LIN {X 0,Y 523.917,Z 214.223,A -85,B 0,C 180,E1 -4816.833,E2 -4816.833} C_VEL
LIN {X 0,Y 523.939,Z 214.219,A -85,B 0,C 180,E1 -4818.907,E2 -4818.907} C_VEL
LIN {X 0,Y 523.916,Z 214.219,A -85,B 0,C 180,E1 -4821.898,E2 -4821.898} C_VEL
LIN {X 0,Y 523.935,Z 214.221,A -85,B 0,C 180,E1 -4824.909,E2 -4824.909} C_VEL
LIN {X 0,Y 523.935,Z 214.217,A -85,B 0,C 180,E1 -4827.68,E2 -4827.68} C_VEL
LIN {X 0,Y 523.954,Z 214.217,A -85,B 0,C 180,E1 -4830.676,E2 -4830.676} C_VEL
LIN {X 0,Y 523.973,Z 214.213,A -85,B 0,C 180,E1 -4833.728,E2 -4833.728} C_VEL
LIN {X 0,Y 523.925,Z 214.217,A -85,B 0,C 180,E1 -4836.27,E2 -4836.27} C_VEL
LIN {X 0,Y 523.945,Z 214.22,A -85,B 0,C 180,E1 -4838.767,E2 -4838.767} C_VEL
LIN {X 0,Y 523.948,Z 214.219,A -85,B 0,C 180,E1 -4841.221,E2 -4841.221} C_VEL
LIN {X 0,Y 523.935,Z 214.217,A -85,B 0,C 180,E1 -4843.639,E2 -4843.639} C_VEL
LIN {X 0,Y 523.939,Z 214.213,A -85,B 0,C 180,E1 -4846.028,E2 -4846.028} C_VEL
LIN {X 0,Y 524.012,Z 214.209,A -85,B 0,C 180,E1 -4848.394,E2 -4848.394} C_VEL
LIN {X 0,Y 524.003,Z 214.209,A -85,B 0,C 180,E1 -4851.516,E2 -4851.516} C_VEL
LIN {X 0,Y 524.08,Z 214.203,A -85,B 0,C 180,E1 -4854.614,E2 -4854.614} C_VEL
LIN {X 0,Y 524.111,Z 214.195,A -85,B 0,C 180,E1 -4857.695,E2 -4857.695} C_VEL
LIN {X 0,Y 524.123,Z 214.199,A -85,B 0,C 180,E1 -4860.768,E2 -4860.768} C_VEL
LIN {X 0,Y 524.069,Z 214.203,A -85,B 0,C 180,E1 -4863.075,E2 -4863.075} C_VEL
LIN {X 0,Y 524.035,Z 214.205,A -85,B 0,C 180,E1 -4866.159,E2 -4866.159} C_VEL
LIN {X 0,Y 524.003,Z 214.212,A -85,B 0,C 180,E1 -4868.484,E2 -4868.484} C_VEL
LIN {X 0,Y 524.002,Z 214.206,A -85,B 0,C 180,E1 -4871.739,E2 -4871.739} C_VEL
LIN {X 0,Y 523.994,Z 214.212,A -85,B 0,C 180,E1 -4875.053,E2 -4875.053} C_VEL
LIN {X 0,Y 523.963,Z 214.214,A -85,B 0,C 180,E1 -4877.969,E2 -4877.969} C_VEL
LIN {X 0,Y 523.971,Z 214.218,A -85,B 0,C 180,E1 -4880.41,E2 -4880.41} C_VEL
LIN {X 0,Y 523.91,Z 214.224,A -85,B 0,C 180,E1 -4882.894,E2 -4882.894} C_VEL
LIN {X 0,Y 523.934,Z 214.217,A -85,B 0,C 180,E1 -4885.42,E2 -4885.42} C_VEL
LIN {X 0,Y 523.917,Z 214.221,A -85,B 0,C 180,E1 -4888.002,E2 -4888.002} C_VEL
LIN {X 0,Y 523.944,Z 214.22,A -85,B 0,C 180,E1 -4890.855,E2 -4890.855} C_VEL
LIN {X 0,Y 523.929,Z 214.22,A -85,B 0,C 180,E1 -4893.73,E2 -4893.73} C_VEL
LIN {X 0,Y 523.888,Z 214.233,A -85,B 0,C 180,E1 -4896.399,E2 -4896.399} C_VEL
LIN {X 0,Y 523.911,Z 214.222,A -85,B 0,C 180,E1 -4899.086,E2 -4899.086} C_VEL
LIN {X 0,Y 523.91,Z 214.226,A -85,B 0,C 180,E1 -4902.123,E2 -4902.123} C_VEL
LIN {X 0,Y 523.982,Z 214.414,A -85,B 0,C 180,E1 -4904.794,E2 -4904.794} C_VEL
LIN {X 0,Y 524.512,Z 219.231,A -85,B 0,C 180,E1 -4905.676,E2 -4905.676} C_VEL
LIN {X 0,Y 523.83,Z 222.403,A -85,B 0,C 180,E1 -4906.215,E2 -4906.215} C_VEL
LIN {X 0,Y 517.981,Z 233.191,A -85,B 0,C 180,E1 -4907.936,E2 -4907.936} C_VEL
LIN {X 0,Y 517.272,Z 236.366,A -85,B 0,C 180,E1 -4908.486,E2 -4908.486} C_VEL
LIN {X 0,Y 517.246,Z 243.207,A -85,B 0,C 180,E1 -4909.693,E2 -4909.693} C_VEL
LIN {X 0,Y 519.105,Z 253.868,A -85,B 0,C 180,E1 -4909.902,E2 -4909.902} C_VEL
LIN {X 0,Y 518.562,Z 350.909,A -85,B 0,C 180,E1 -4911.278,E2 -4911.278} C_VEL
LIN {X 0,Y 518.36,Z 364.692,A -85,B 0,C 180,E1 -4911.649,E2 -4911.649} C_VEL
LIN {X 0,Y 518.235,Z 376.182,A -85,B 0,C 180,E1 -4912.107,E2 -4912.107} C_VEL
LIN {X 0,Y 517.887,Z 387.78,A -85,B 0,C 180,E1 -4912.719,E2 -4912.719} C_VEL
LIN {X 0,Y 517.552,Z 399.902,A -85,B 0,C 180,E1 -4913.552,E2 -4913.552} C_VEL
LIN {X 0,Y 517.263,Z 410.497,A -85,B 0,C 180,E1 -4914.47,E2 -4914.47} C_VEL
LIN {X 0,Y 516.988,Z 419.34,A -85,B 0,C 180,E1 -4915.418,E2 -4915.418} C_VEL
LIN {X 0,Y 516.757,Z 428.136,A -85,B 0,C 180,E1 -4916.578,E2 -4916.578} C_VEL
LIN {X 0,Y 516.601,Z 435.226,A -85,B 0,C 180,E1 -4917.734,E2 -4917.734} C_VEL
LIN {X 0,Y 516.454,Z 441.481,A -85,B 0,C 180,E1 -4919.017,E2 -4919.017} C_VEL
LIN {X 0,Y 516.351,Z 445.996,A -85,B 0,C 180,E1 -4920.211,E2 -4920.211} C_VEL
LIN {X 0,Y 516.251,Z 449.73,A -85,B 0,C 180,E1 -4921.545,E2 -4921.545} C_VEL
LIN {X 0,Y 516.202,Z 451.517,A -85,B 0,C 180,E1 -4922.425,E2 -4922.425} C_VEL
LIN {X 0,Y 516.185,Z 452.756,A -85,B 0,C 180,E1 -4923.301,E2 -4923.301} C_VEL
LIN {X 0,Y 516.175,Z 453.484,A -85,B 0,C 180,E1 -4924.17,E2 -4924.17} C_VEL
LIN {X 0,Y 516.152,Z 453.754,A -85,B 0,C 180,E1 -4925.033,E2 -4925.033} C_VEL
LIN {X 0,Y 516.161,Z 453.498,A -85,B 0,C 180,E1 -4925.891,E2 -4925.891} C_VEL
LIN {X 0,Y 516.148,Z 452.797,A -85,B 0,C 180,E1 -4926.742,E2 -4926.742} C_VEL
LIN {X 0,Y 516.194,Z 451.266,A -85,B 0,C 180,E1 -4927.793,E2 -4927.793} C_VEL
LIN {X 0,Y 516.328,Z 447.84,A -85,B 0,C 180,E1 -4929.274,E2 -4929.274} C_VEL
LIN {X 0,Y 516.413,Z 443.693,A -85,B 0,C 180,E1 -4930.523,E2 -4930.523} C_VEL
LIN {X 0,Y 516.522,Z 438.291,A -85,B 0,C 180,E1 -4931.763,E2 -4931.763} C_VEL
LIN {X 0,Y 516.657,Z 431.466,A -85,B 0,C 180,E1 -4932.995,E2 -4932.995} C_VEL
LIN {X 0,Y 516.9,Z 422.964,A -85,B 0,C 180,E1 -4934.221,E2 -4934.221} C_VEL
LIN {X 0,Y 517.139,Z 414.239,A -85,B 0,C 180,E1 -4935.237,E2 -4935.237} C_VEL
LIN {X 0,Y 517.457,Z 403.416,A -85,B 0,C 180,E1 -4936.25,E2 -4936.25} C_VEL
LIN {X 0,Y 517.781,Z 392.651,A -85,B 0,C 180,E1 -4937.058,E2 -4937.058} C_VEL
LIN {X 0,Y 518.107,Z 381.878,A -85,B 0,C 180,E1 -4937.701,E2 -4937.701} C_VEL
LIN {X 0,Y 518.31,Z 369.482,A -85,B 0,C 180,E1 -4938.265,E2 -4938.265} C_VEL
LIN {X 0,Y 518.488,Z 357.153,A -85,B 0,C 180,E1 -4938.665,E2 -4938.665} C_VEL
LIN {X 0,Y 518.618,Z 345.034,A -85,B 0,C 180,E1 -4938.915,E2 -4938.915} C_VEL
LIN {X 0,Y 518.976,Z 252.872,A -85,B 0,C 180,E1 -4940.205,E2 -4940.205} C_VEL
LIN {X 0,Y 517.248,Z 243.012,A -85,B 0,C 180,E1 -4940.419,E2 -4940.419} C_VEL
LIN {X 0,Y 517.558,Z 226.28,A -85,B 0,C 180,E1 -4943.568,E2 -4943.568} C_VEL
LIN {X 0,Y 517.515,Z 219.114,A -85,B 0,C 180,E1 -4944.936,E2 -4944.936} C_VEL
LIN {X 0,Y 516.921,Z 215.099,A -85,B 0,C 180,E1 -4945.76,E2 -4945.76} C_VEL
LIN {X 0,Y 517.077,Z 215.08,A -85,B 0,C 180,E1 -4947.663,E2 -4947.663} C_VEL
LIN {X 0,Y 517.069,Z 215.077,A -85,B 0,C 180,E1 -4950,E2 -4950} C_VEL
LIN {X 0,Y 517.077,Z 215.072,A -85,B 0,C 180,E1 -4952.337,E2 -4952.337} C_VEL
LIN {X 0,Y 516.978,Z 215.085,A -85,B 0,C 180,E1 -4956.243,E2 -4956.243} C_VEL
LIN {X 0,Y 516.94,Z 215.093,A -85,B 0,C 180,E1 -4959.389,E2 -4959.389} C_VEL
LIN {X 0,Y 516.955,Z 215.092,A -85,B 0,C 180,E1 -4961.807,E2 -4961.807} C_VEL
LIN {X 0,Y 516.942,Z 215.091,A -85,B 0,C 180,E1 -4965.144,E2 -4965.144} C_VEL
LIN {X 0,Y 516.881,Z 215.097,A -85,B 0,C 180,E1 -4968.224,E2 -4968.224} C_VEL
LIN {X 0,Y 516.907,Z 215.093,A -85,B 0,C 180,E1 -4970.701,E2 -4970.701} C_VEL
LIN {X 0,Y 516.887,Z 215.097,A -85,B 0,C 180,E1 -4974.073,E2 -4974.073} C_VEL
LIN {X 0,Y 516.897,Z 215.094,A -85,B 0,C 180,E1 -4976.659,E2 -4976.659} C_VEL
LIN {X 0,Y 516.91,Z 215.1,A -85,B 0,C 180,E1 -4979.523,E2 -4979.523} C_VEL
LIN {X 0,Y 516.897,Z 215.094,A -85,B 0,C 180,E1 -4982.543,E2 -4982.543} C_VEL
LIN {X 0,Y 516.864,Z 215.104,A -85,B 0,C 180,E1 -4985.329,E2 -4985.329} C_VEL
LIN {X 0,Y 516.878,Z 215.099,A -85,B 0,C 180,E1 -4987.942,E2 -4987.942} C_VEL
LIN {X 0,Y 516.882,Z 215.098,A -85,B 0,C 180,E1 -4990.741,E2 -4990.741} C_VEL
LIN {X 0,Y 516.881,Z 215.099,A -85,B 0,C 180,E1 -4993.903,E2 -4993.903} C_VEL
LIN {X 0,Y 516.881,Z 215.097,A -85,B 0,C 180,E1 -4996.107,E2 -4996.107} C_VEL
LIN {X 0,Y 516.912,Z 215.093,A -85,B 0,C 180,E1 -4998.398,E2 -4998.398} C_VEL
LIN {X 0,Y 516.879,Z 215.102,A -85,B 0,C 180,E1 -5001.284,E2 -5001.284} C_VEL
LIN {X 0,Y 516.887,Z 215.096,A -85,B 0,C 180,E1 -5004.221,E2 -5004.221} C_VEL
LIN {X 0,Y 516.893,Z 215.1,A -85,B 0,C 180,E1 -5007.053,E2 -5007.053} C_VEL
LIN {X 0,Y 516.89,Z 215.098,A -85,B 0,C 180,E1 -5009.796,E2 -5009.796} C_VEL
LIN {X 0,Y 516.924,Z 215.092,A -85,B 0,C 180,E1 -5012.467,E2 -5012.467} C_VEL
LIN {X 0,Y 516.909,Z 215.098,A -85,B 0,C 180,E1 -5015.072,E2 -5015.072} C_VEL
LIN {X 0,Y 516.868,Z 215.102,A -85,B 0,C 180,E1 -5017.621,E2 -5017.621} C_VEL
LIN {X 0,Y 516.929,Z 215.091,A -85,B 0,C 180,E1 -5020.13,E2 -5020.13} C_VEL
LIN {X 0,Y 516.919,Z 215.094,A -85,B 0,C 180,E1 -5022.596,E2 -5022.596} C_VEL
LIN {X 0,Y 516.94,Z 215.095,A -85,B 0,C 180,E1 -5025.03,E2 -5025.03} C_VEL
LIN {X 0,Y 516.963,Z 215.087,A -85,B 0,C 180,E1 -5028.233,E2 -5028.233} C_VEL
LIN {X 0,Y 516.967,Z 215.091,A -85,B 0,C 180,E1 -5031.4,E2 -5031.4} C_VEL
LIN {X 0,Y 517.013,Z 215.081,A -85,B 0,C 180,E1 -5033.757,E2 -5033.757} C_VEL
LIN {X 0,Y 517.083,Z 215.073,A -85,B 0,C 180,E1 -5037.663,E2 -5037.663} C_VEL
LIN {X 0,Y 517.09,Z 215.077,A -85,B 0,C 180,E1 -5040.779,E2 -5040.779} C_VEL
LIN {X 0,Y 517.01,Z 215.086,A -85,B 0,C 180,E1 -5043.117,E2 -5043.117} C_VEL
LIN {X 0,Y 517.013,Z 215.081,A -85,B 0,C 180,E1 -5046.243,E2 -5046.243} C_VEL
LIN {X 0,Y 516.949,Z 215.091,A -85,B 0,C 180,E1 -5049.389,E2 -5049.389} C_VEL
LIN {X 0,Y 516.949,Z 215.088,A -85,B 0,C 180,E1 -5051.807,E2 -5051.807} C_VEL
LIN {X 0,Y 516.942,Z 215.094,A -85,B 0,C 180,E1 -5055.147,E2 -5055.147} C_VEL
LIN {X 0,Y 516.923,Z 215.093,A -85,B 0,C 180,E1 -5058.222,E2 -5058.222} C_VEL
LIN {X 0,Y 516.91,Z 215.1,A -85,B 0,C 180,E1 -5060.702,E2 -5060.702} C_VEL
LIN {X 0,Y 516.909,Z 215.093,A -85,B 0,C 180,E1 -5064.072,E2 -5064.072} C_VEL
LIN {X 0,Y 516.922,Z 215.098,A -85,B 0,C 180,E1 -5066.658,E2 -5066.658} C_VEL
LIN {X 0,Y 516.909,Z 215.094,A -85,B 0,C 180,E1 -5069.524,E2 -5069.524} C_VEL
LIN {X 0,Y 516.893,Z 215.1,A -85,B 0,C 180,E1 -5072.544,E2 -5072.544} C_VEL
LIN {X 0,Y 516.878,Z 215.098,A -85,B 0,C 180,E1 -5075.332,E2 -5075.332} C_VEL
LIN {X 0,Y 516.879,Z 215.097,A -85,B 0,C 180,E1 -5077.943,E2 -5077.943} C_VEL
LIN {X 0,Y 516.881,Z 215.103,A -85,B 0,C 180,E1 -5080.742,E2 -5080.742} C_VEL
LIN {X 0,Y 516.881,Z 215.101,A -85,B 0,C 180,E1 -5082.832,E2 -5082.832} C_VEL
LIN {X 0,Y 516.922,Z 215.095,A -85,B 0,C 180,E1 -5085.01,E2 -5085.01} C_VEL
LIN {X 0,Y 516.912,Z 215.097,A -85,B 0,C 180,E1 -5088.399,E2 -5088.399} C_VEL
LIN {X 0,Y 516.879,Z 215.097,A -85,B 0,C 180,E1 -5091.284,E2 -5091.284} C_VEL
LIN {X 0,Y 516.867,Z 215.101,A -85,B 0,C 180,E1 -5094.22,E2 -5094.22} C_VEL
LIN {X 0,Y 516.895,Z 215.096,A -85,B 0,C 180,E1 -5097.053,E2 -5097.053} C_VEL
LIN {X 0,Y 516.892,Z 215.096,A -85,B 0,C 180,E1 -5099.797,E2 -5099.797} C_VEL
LIN {X 0,Y 516.921,Z 215.1,A -85,B 0,C 180,E1 -5102.467,E2 -5102.467} C_VEL
LIN {X 0,Y 516.917,Z 215.221,A -85,B 0,C 180,E1 -5105.707,E2 -5105.707} C_VEL
LIN {X 0,Y 518.391,Z 223.809,A -85,B 0,C 180,E1 -5107.206,E2 -5107.206} C_VEL
LIN {X 0,Y 518.01,Z 239.597,A -85,B 0,C 180,E1 -5109.786,E2 -5109.786} C_VEL
LIN {X 0,Y 517.505,Z 258.465,A -85,B 0,C 180,E1 -5112.82,E2 -5112.82} C_VEL
LIN {X 0,Y 517.274,Z 269.995,A -85,B 0,C 180,E1 -5114.637,E2 -5114.637} C_VEL
LIN {X 0,Y 519.058,Z 282.247,A -85,B 0,C 180,E1 -5114.864,E2 -5114.864} C_VEL
LIN {X 0,Y 518.575,Z 377.579,A -85,B 0,C 180,E1 -5116.206,E2 -5116.206} C_VEL
LIN {X 0,Y 518.325,Z 390.991,A -85,B 0,C 180,E1 -5116.549,E2 -5116.549} C_VEL
LIN {X 0,Y 518.06,Z 404.352,A -85,B 0,C 180,E1 -5117.066,E2 -5117.066} C_VEL
LIN {X 0,Y 517.79,Z 416.6,A -85,B 0,C 180,E1 -5117.722,E2 -5117.722} C_VEL
LIN {X 0,Y 517.515,Z 428.485,A -85,B 0,C 180,E1 -5118.544,E2 -5118.544} C_VEL
LIN {X 0,Y 517.176,Z 438.705,A -85,B 0,C 180,E1 -5119.429,E2 -5119.429} C_VEL
LIN {X 0,Y 516.914,Z 447.896,A -85,B 0,C 180,E1 -5120.413,E2 -5120.413} C_VEL
LIN {X 0,Y 516.664,Z 456.848,A -85,B 0,C 180,E1 -5121.592,E2 -5121.592} C_VEL
LIN {X 0,Y 516.504,Z 464.055,A -85,B 0,C 180,E1 -5122.77,E2 -5122.77} C_VEL
LIN {X 0,Y 516.416,Z 470.617,A -85,B 0,C 180,E1 -5124.142,E2 -5124.142} C_VEL
LIN {X 0,Y 516.268,Z 474.954,A -85,B 0,C 180,E1 -5125.315,E2 -5125.315} C_VEL
LIN {X 0,Y 516.352,Z 477.254,A -85,B 0,C 180,E1 -5126.098,E2 -5126.098} C_VEL
LIN {X 0,Y 516.282,Z 479.114,A -85,B 0,C 180,E1 -5126.879,E2 -5126.879} C_VEL
LIN {X 0,Y 516.261,Z 480.509,A -85,B 0,C 180,E1 -5127.66,E2 -5127.66} C_VEL
LIN {X 0,Y 516.161,Z 482.109,A -85,B 0,C 180,E1 -5129.22,E2 -5129.22} C_VEL
LIN {X 0,Y 516.157,Z 482.325,A -85,B 0,C 180,E1 -5130,E2 -5130} C_VEL
LIN {X 0,Y 516.192,Z 481.5,A -85,B 0,C 180,E1 -5131.56,E2 -5131.56} C_VEL
LIN {X 0,Y 516.261,Z 480.504,A -85,B 0,C 180,E1 -5132.341,E2 -5132.341} C_VEL
LIN {X 0,Y 516.282,Z 479.107,A -85,B 0,C 180,E1 -5133.121,E2 -5133.121} C_VEL
LIN {X 0,Y 516.311,Z 476.168,A -85,B 0,C 180,E1 -5134.294,E2 -5134.294} C_VEL
LIN {X 0,Y 516.374,Z 472.189,A -85,B 0,C 180,E1 -5135.467,E2 -5135.467} C_VEL
LIN {X 0,Y 516.422,Z 466.989,A -85,B 0,C 180,E1 -5136.659,E2 -5136.659} C_VEL
LIN {X 0,Y 516.575,Z 460.619,A -85,B 0,C 180,E1 -5137.819,E2 -5137.819} C_VEL
LIN {X 0,Y 516.769,Z 452.576,A -85,B 0,C 180,E1 -5138.998,E2 -5138.998} C_VEL
LIN {X 0,Y 516.978,Z 444.378,A -85,B 0,C 180,E1 -5139.981,E2 -5139.981} C_VEL
LIN {X 0,Y 517.318,Z 434.382,A -85,B 0,C 180,E1 -5140.964,E2 -5140.964} C_VEL
LIN {X 0,Y 517.604,Z 424.513,A -85,B 0,C 180,E1 -5141.752,E2 -5141.752} C_VEL
LIN {X 0,Y 517.845,Z 413.377,A -85,B 0,C 180,E1 -5142.465,E2 -5142.465} C_VEL
LIN {X 0,Y 518.135,Z 400.872,A -85,B 0,C 180,E1 -5143.082,E2 -5143.082} C_VEL
LIN {X 0,Y 518.42,Z 388.59,A -85,B 0,C 180,E1 -5143.524,E2 -5143.524} C_VEL
LIN {X 0,Y 518.61,Z 376.024,A -85,B 0,C 180,E1 -5143.819,E2 -5143.819} C_VEL
LIN {X 0,Y 518.926,Z 280.302,A -85,B 0,C 180,E1 -5145.166,E2 -5145.166} C_VEL
LIN {X 0,Y 517.239,Z 269.533,A -85,B 0,C 180,E1 -5145.393,E2 -5145.393} C_VEL
LIN {X 0,Y 517.719,Z 249.263,A -85,B 0,C 180,E1 -5148.603,E2 -5148.603} C_VEL
LIN {X 0,Y 518.131,Z 231.305,A -85,B 0,C 180,E1 -5151.483,E2 -5151.483} C_VEL
LIN {X 0,Y 518.241,Z 222.553,A -85,B 0,C 180,E1 -5152.907,E2 -5152.907} C_VEL
LIN {X 0,Y 516.907,Z 215.098,A -85,B 0,C 180,E1 -5154.223,E2 -5154.223} C_VEL
LIN {X 0,Y 516.922,Z 215.098,A -85,B 0,C 180,E1 -5157.533,E2 -5157.533} C_VEL
LIN {X 0,Y 516.888,Z 215.096,A -85,B 0,C 180,E1 -5160.204,E2 -5160.204} C_VEL
LIN {X 0,Y 516.896,Z 215.099,A -85,B 0,C 180,E1 -5162.947,E2 -5162.947} C_VEL
LIN {X 0,Y 516.869,Z 215.1,A -85,B 0,C 180,E1 -5165.78,E2 -5165.78} C_VEL
LIN {X 0,Y 516.88,Z 215.097,A -85,B 0,C 180,E1 -5168.716,E2 -5168.716} C_VEL
LIN {X 0,Y 516.912,Z 215.094,A -85,B 0,C 180,E1 -5171.775,E2 -5171.775} C_VEL
LIN {X 0,Y 516.923,Z 215.096,A -85,B 0,C 180,E1 -5175.01,E2 -5175.01} C_VEL
LIN {X 0,Y 516.913,Z 215.09,A -85,B 0,C 180,E1 -5178.399,E2 -5178.399} C_VEL
LIN {X 0,Y 516.88,Z 215.102,A -85,B 0,C 180,E1 -5181.284,E2 -5181.284} C_VEL
LIN {X 0,Y 516.888,Z 215.094,A -85,B 0,C 180,E1 -5184.221,E2 -5184.221} C_VEL
LIN {X 0,Y 516.894,Z 215.101,A -85,B 0,C 180,E1 -5187.053,E2 -5187.053} C_VEL
LIN {X 0,Y 516.891,Z 215.095,A -85,B 0,C 180,E1 -5189.796,E2 -5189.796} C_VEL
LIN {X 0,Y 516.925,Z 215.089,A -85,B 0,C 180,E1 -5192.467,E2 -5192.467} C_VEL
LIN {X 0,Y 516.908,Z 215.1,A -85,B 0,C 180,E1 -5195.072,E2 -5195.072} C_VEL
LIN {X 0,Y 516.884,Z 215.096,A -85,B 0,C 180,E1 -5198.462,E2 -5198.462} C_VEL
LIN {X 0,Y 516.901,Z 215.099,A -85,B 0,C 180,E1 -5200.955,E2 -5200.955} C_VEL
LIN {X 0,Y 516.912,Z 215.094,A -85,B 0,C 180,E1 -5203.41,E2 -5203.41} C_VEL
LIN {X 0,Y 516.894,Z 215.09,A -85,B 0,C 180,E1 -5205.834,E2 -5205.834} C_VEL
LIN {X 0,Y 516.965,Z 215.085,A -85,B 0,C 180,E1 -5208.234,E2 -5208.234} C_VEL
LIN {X 0,Y 516.968,Z 215.086,A -85,B 0,C 180,E1 -5211.4,E2 -5211.4} C_VEL
LIN {X 0,Y 517.002,Z 215.08,A -85,B 0,C 180,E1 -5213.757,E2 -5213.757} C_VEL
LIN {X 0,Y 517.012,Z 215.087,A -85,B 0,C 180,E1 -5216.883,E2 -5216.883} C_VEL
LIN {X 0,Y 517.085,Z 215.067,A -85,B 0,C 180,E1 -5220,E2 -5220} C_VEL
LIN {X 0,Y 517.01,Z 215.081,A -85,B 0,C 180,E1 -5223.117,E2 -5223.117} C_VEL
LIN {X 0,Y 517.001,Z 215.083,A -85,B 0,C 180,E1 -5226.243,E2 -5226.243} C_VEL
LIN {X 0,Y 516.951,Z 215.088,A -85,B 0,C 180,E1 -5229.389,E2 -5229.389} C_VEL
LIN {X 0,Y 516.951,Z 215.085,A -85,B 0,C 180,E1 -5231.807,E2 -5231.807} C_VEL
LIN {X 0,Y 516.947,Z 215.089,A -85,B 0,C 180,E1 -5235.148,E2 -5235.148} C_VEL
LIN {X 0,Y 516.924,Z 215.093,A -85,B 0,C 180,E1 -5238.222,E2 -5238.222} C_VEL
LIN {X 0,Y 516.912,Z 215.099,A -85,B 0,C 180,E1 -5240.702,E2 -5240.702} C_VEL
LIN {X 0,Y 516.901,Z 215.095,A -85,B 0,C 180,E1 -5244.073,E2 -5244.073} C_VEL
LIN {X 0,Y 516.896,Z 215.102,A -85,B 0,C 180,E1 -5246.66,E2 -5246.66} C_VEL
LIN {X 0,Y 516.909,Z 215.09,A -85,B 0,C 180,E1 -5249.524,E2 -5249.524} C_VEL
LIN {X 0,Y 516.894,Z 215.1,A -85,B 0,C 180,E1 -5252.543,E2 -5252.543} C_VEL
LIN {X 0,Y 516.861,Z 215.1,A -85,B 0,C 180,E1 -5255.329,E2 -5255.329} C_VEL
LIN {X 0,Y 516.874,Z 215.103,A -85,B 0,C 180,E1 -5258.717,E2 -5258.717} C_VEL
LIN {X 0,Y 516.884,Z 215.098,A -85,B 0,C 180,E1 -5261.778,E2 -5261.778} C_VEL
LIN {X 0,Y 516.939,Z 215.185,A -85,B 0,C 180,E1 -5264.645,E2 -5264.645} C_VEL
LIN {X 0,Y 517.539,Z 220.322,A -85,B 0,C 180,E1 -5265.603,E2 -5265.603} C_VEL
LIN {X 0,Y 517.284,Z 235.631,A -85,B 0,C 180,E1 -5268.353,E2 -5268.353} C_VEL
LIN {X 0,Y 517.272,Z 236.366,A -85,B 0,C 180,E1 -5268.486,E2 -5268.486} C_VEL
LIN {X 0,Y 517.024,Z 238.776,A -85,B 0,C 180,E1 -5268.821,E2 -5268.821} C_VEL
LIN {X 0,Y 516.069,Z 243.375,A -85,B 0,C 180,E1 -5269.209,E2 -5269.209} C_VEL
LIN {X 0,Y 514.786,Z 248.632,A -85,B 0,C 180,E1 -5269.477,E2 -5269.477} C_VEL
LIN {X 0,Y 513.088,Z 256.44,A -85,B 0,C 180,E1 -5269.707,E2 -5269.707} C_VEL
LIN {X 0,Y 512.279,Z 264.548,A -85,B 0,C 180,E1 -5269.845,E2 -5269.845} C_VEL
LIN {X 0,Y 511.674,Z 350.916,A -85,B 0,C 180,E1 -5271.086,E2 -5271.086} C_VEL
LIN {X 0,Y 511.469,Z 364.681,A -85,B 0,C 180,E1 -5271.459,E2 -5271.459} C_VEL
LIN {X 0,Y 511.308,Z 377.409,A -85,B 0,C 180,E1 -5271.979,E2 -5271.979} C_VEL
LIN {X 0,Y 510.931,Z 389.246,A -85,B 0,C 180,E1 -5272.631,E2 -5272.631} C_VEL
LIN {X 0,Y 510.57,Z 400.988,A -85,B 0,C 180,E1 -5273.464,E2 -5273.464} C_VEL
LIN {X 0,Y 510.259,Z 410.983,A -85,B 0,C 180,E1 -5274.354,E2 -5274.354} C_VEL
LIN {X 0,Y 509.969,Z 420.108,A -85,B 0,C 180,E1 -5275.356,E2 -5275.356} C_VEL
LIN {X 0,Y 509.704,Z 428.787,A -85,B 0,C 180,E1 -5276.528,E2 -5276.528} C_VEL
LIN {X 0,Y 509.557,Z 435.759,A -85,B 0,C 180,E1 -5277.693,E2 -5277.693} C_VEL
LIN {X 0,Y 509.381,Z 442.17,A -85,B 0,C 180,E1 -5279.055,E2 -5279.055} C_VEL
LIN {X 0,Y 509.24,Z 446.982,A -85,B 0,C 180,E1 -5280.397,E2 -5280.397} C_VEL
LIN {X 0,Y 509.181,Z 450.077,A -85,B 0,C 180,E1 -5281.563,E2 -5281.563} C_VEL
LIN {X 0,Y 509.084,Z 452.479,A -85,B 0,C 180,E1 -5282.898,E2 -5282.898} C_VEL
LIN {X 0,Y 509.085,Z 453.471,A -85,B 0,C 180,E1 -5283.811,E2 -5283.811} C_VEL
LIN {X 0,Y 509.053,Z 453.881,A -85,B 0,C 180,E1 -5284.66,E2 -5284.66} C_VEL
LIN {X 0,Y 509.056,Z 453.825,A -85,B 0,C 180,E1 -5285.671,E2 -5285.671} C_VEL
LIN {X 0,Y 509.054,Z 453.363,A -85,B 0,C 180,E1 -5286.399,E2 -5286.399} C_VEL
LIN {X 0,Y 509.107,Z 451.782,A -85,B 0,C 180,E1 -5287.655,E2 -5287.655} C_VEL
LIN {X 0,Y 509.269,Z 447.861,A -85,B 0,C 180,E1 -5289.397,E2 -5289.397} C_VEL
LIN {X 0,Y 509.339,Z 443.653,A -85,B 0,C 180,E1 -5290.661,E2 -5290.661} C_VEL
LIN {X 0,Y 509.475,Z 438.391,A -85,B 0,C 180,E1 -5291.874,E2 -5291.874} C_VEL
LIN {X 0,Y 509.61,Z 431.282,A -85,B 0,C 180,E1 -5293.165,E2 -5293.165} C_VEL
LIN {X 0,Y 509.862,Z 424.075,A -85,B 0,C 180,E1 -5294.223,E2 -5294.223} C_VEL
LIN {X 0,Y 510.108,Z 415.736,A -85,B 0,C 180,E1 -5295.233,E2 -5295.233} C_VEL
LIN {X 0,Y 510.434,Z 406.44,A -85,B 0,C 180,E1 -5296.159,E2 -5296.159} C_VEL
LIN {X 0,Y 510.707,Z 396.352,A -85,B 0,C 180,E1 -5296.977,E2 -5296.977} C_VEL
LIN {X 0,Y 511.079,Z 385.317,A -85,B 0,C 180,E1 -5297.691,E2 -5297.691} C_VEL
LIN {X 0,Y 511.37,Z 373.078,A -85,B 0,C 180,E1 -5298.304,E2 -5298.304} C_VEL
LIN {X 0,Y 511.574,Z 360.595,A -85,B 0,C 180,E1 -5298.761,E2 -5298.761} C_VEL
LIN {X 0,Y 511.718,Z 347.59,A -85,B 0,C 180,E1 -5299.065,E2 -5299.065} C_VEL
LIN {X 0,Y 512.177,Z 253.988,A -85,B 0,C 180,E1 -5300.398,E2 -5300.398} C_VEL
LIN {X 0,Y 510.25,Z 243.18,A -85,B 0,C 180,E1 -5300.636,E2 -5300.636} C_VEL
LIN {X 0,Y 510.579,Z 227.192,A -85,B 0,C 180,E1 -5303.678,E2 -5303.678} C_VEL
LIN {X 0,Y 510.612,Z 221,A -85,B 0,C 180,E1 -5304.867,E2 -5304.867} C_VEL
LIN {X 0,Y 509.861,Z 215.978,A -85,B 0,C 180,E1 -5305.899,E2 -5305.899} C_VEL
LIN {X 0,Y 510.045,Z 215.955,A -85,B 0,C 180,E1 -5307.631,E2 -5307.631} C_VEL
LIN {X 0,Y 510.038,Z 215.953,A -85,B 0,C 180,E1 -5310,E2 -5310} C_VEL
LIN {X 0,Y 510.046,Z 215.947,A -85,B 0,C 180,E1 -5312.369,E2 -5312.369} C_VEL
LIN {X 0,Y 509.944,Z 215.966,A -85,B 0,C 180,E1 -5315.536,E2 -5315.536} C_VEL
LIN {X 0,Y 509.904,Z 215.965,A -85,B 0,C 180,E1 -5318.72,E2 -5318.72} C_VEL
LIN {X 0,Y 509.907,Z 215.968,A -85,B 0,C 180,E1 -5321.931,E2 -5321.931} C_VEL
LIN {X 0,Y 509.898,Z 215.969,A -85,B 0,C 180,E1 -5325.241,E2 -5325.241} C_VEL
LIN {X 0,Y 509.84,Z 215.973,A -85,B 0,C 180,E1 -5328.484,E2 -5328.484} C_VEL
LIN {X 0,Y 509.848,Z 215.974,A -85,B 0,C 180,E1 -5331.001,E2 -5331.001} C_VEL
LIN {X 0,Y 509.821,Z 215.983,A -85,B 0,C 180,E1 -5333.564,E2 -5333.564} C_VEL
LIN {X 0,Y 509.877,Z 215.969,A -85,B 0,C 180,E1 -5336.37,E2 -5336.37} C_VEL
LIN {X 0,Y 509.853,Z 215.973,A -85,B 0,C 180,E1 -5338.845,E2 -5338.845} C_VEL
LIN {X 0,Y 509.821,Z 215.983,A -85,B 0,C 180,E1 -5341.59,E2 -5341.59} C_VEL
LIN {X 0,Y 509.847,Z 215.973,A -85,B 0,C 180,E1 -5344.413,E2 -5344.413} C_VEL
LIN {X 0,Y 509.808,Z 215.983,A -85,B 0,C 180,E1 -5347.341,E2 -5347.341} C_VEL
LIN {X 0,Y 509.838,Z 215.974,A -85,B 0,C 180,E1 -5350.382,E2 -5350.382} C_VEL
LIN {X 0,Y 509.804,Z 215.982,A -85,B 0,C 180,E1 -5353.059,E2 -5353.059} C_VEL
LIN {X 0,Y 509.822,Z 215.979,A -85,B 0,C 180,E1 -5355.793,E2 -5355.793} C_VEL
LIN {X 0,Y 509.854,Z 215.973,A -85,B 0,C 180,E1 -5358.574,E2 -5358.574} C_VEL
LIN {X 0,Y 509.849,Z 215.975,A -85,B 0,C 180,E1 -5361.786,E2 -5361.786} C_VEL
LIN {X 0,Y 509.842,Z 215.975,A -85,B 0,C 180,E1 -5364.623,E2 -5364.623} C_VEL
LIN {X 0,Y 509.859,Z 215.977,A -85,B 0,C 180,E1 -5367.48,E2 -5367.48} C_VEL
LIN {X 0,Y 509.857,Z 215.972,A -85,B 0,C 180,E1 -5370.273,E2 -5370.273} C_VEL
LIN {X 0,Y 509.881,Z 215.973,A -85,B 0,C 180,E1 -5372.944,E2 -5372.944} C_VEL
LIN {X 0,Y 509.868,Z 215.974,A -85,B 0,C 180,E1 -5375.574,E2 -5375.574} C_VEL
LIN {X 0,Y 509.82,Z 215.977,A -85,B 0,C 180,E1 -5378.148,E2 -5378.148} C_VEL
LIN {X 0,Y 509.86,Z 215.974,A -85,B 0,C 180,E1 -5380.681,E2 -5380.681} C_VEL
LIN {X 0,Y 509.88,Z 215.974,A -85,B 0,C 180,E1 -5383.174,E2 -5383.174} C_VEL
LIN {X 0,Y 509.861,Z 215.974,A -85,B 0,C 180,E1 -5385.634,E2 -5385.634} C_VEL
LIN {X 0,Y 509.911,Z 215.971,A -85,B 0,C 180,E1 -5388.874,E2 -5388.874} C_VEL
LIN {X 0,Y 509.949,Z 215.961,A -85,B 0,C 180,E1 -5392.078,E2 -5392.078} C_VEL
LIN {X 0,Y 509.982,Z 215.958,A -85,B 0,C 180,E1 -5394.464,E2 -5394.464} C_VEL
LIN {X 0,Y 510.053,Z 215.949,A -85,B 0,C 180,E1 -5397.631,E2 -5397.631} C_VEL
LIN {X 0,Y 510.06,Z 215.953,A -85,B 0,C 180,E1 -5400.789,E2 -5400.789} C_VEL
LIN {X 0,Y 509.953,Z 215.964,A -85,B 0,C 180,E1 -5403.16,E2 -5403.16} C_VEL
LIN {X 0,Y 509.98,Z 215.958,A -85,B 0,C 180,E1 -5406.33,E2 -5406.33} C_VEL
LIN {X 0,Y 509.912,Z 215.971,A -85,B 0,C 180,E1 -5408.72,E2 -5408.72} C_VEL
LIN {X 0,Y 509.901,Z 215.966,A -85,B 0,C 180,E1 -5411.932,E2 -5411.932} C_VEL
LIN {X 0,Y 509.891,Z 215.971,A -85,B 0,C 180,E1 -5415.242,E2 -5415.242} C_VEL
LIN {X 0,Y 509.886,Z 215.968,A -85,B 0,C 180,E1 -5418.001,E2 -5418.001} C_VEL
LIN {X 0,Y 509.848,Z 215.977,A -85,B 0,C 180,E1 -5421.002,E2 -5421.002} C_VEL
LIN {X 0,Y 509.834,Z 215.975,A -85,B 0,C 180,E1 -5423.563,E2 -5423.563} C_VEL
LIN {X 0,Y 509.908,Z 215.968,A -85,B 0,C 180,E1 -5426.379,E2 -5426.379} C_VEL
LIN {X 0,Y 509.874,Z 215.975,A -85,B 0,C 180,E1 -5428.844,E2 -5428.844} C_VEL
LIN {X 0,Y 509.817,Z 215.977,A -85,B 0,C 180,E1 -5431.59,E2 -5431.59} C_VEL
LIN {X 0,Y 509.85,Z 215.976,A -85,B 0,C 180,E1 -5434.414,E2 -5434.414} C_VEL
LIN {X 0,Y 509.817,Z 215.978,A -85,B 0,C 180,E1 -5437.341,E2 -5437.341} C_VEL
LIN {X 0,Y 509.836,Z 215.978,A -85,B 0,C 180,E1 -5440.383,E2 -5440.383} C_VEL
LIN {X 0,Y 509.821,Z 215.979,A -85,B 0,C 180,E1 -5443.062,E2 -5443.062} C_VEL
LIN {X 0,Y 509.829,Z 215.974,A -85,B 0,C 180,E1 -5445.793,E2 -5445.793} C_VEL
LIN {X 0,Y 509.854,Z 215.979,A -85,B 0,C 180,E1 -5448.575,E2 -5448.575} C_VEL
LIN {X 0,Y 509.849,Z 215.972,A -85,B 0,C 180,E1 -5451.787,E2 -5451.787} C_VEL
LIN {X 0,Y 509.827,Z 215.982,A -85,B 0,C 180,E1 -5454.622,E2 -5454.622} C_VEL
LIN {X 0,Y 509.861,Z 215.97,A -85,B 0,C 180,E1 -5457.481,E2 -5457.481} C_VEL
LIN {X 0,Y 509.859,Z 215.976,A -85,B 0,C 180,E1 -5460.274,E2 -5460.274} C_VEL
LIN {X 0,Y 509.872,Z 215.976,A -85,B 0,C 180,E1 -5462.944,E2 -5462.944} C_VEL
LIN {X 0,Y 509.845,Z 216.014,A -85,B 0,C 180,E1 -5465.514,E2 -5465.514} C_VEL
LIN {X 0,Y 511.46,Z 225.23,A -85,B 0,C 180,E1 -5467.148,E2 -5467.148} C_VEL
LIN {X 0,Y 510.976,Z 241.789,A -85,B 0,C 180,E1 -5469.889,E2 -5469.889} C_VEL
LIN {X 0,Y 510.487,Z 259.54,A -85,B 0,C 180,E1 -5472.783,E2 -5472.783} C_VEL
LIN {X 0,Y 510.264,Z 269.737,A -85,B 0,C 180,E1 -5474.42,E2 -5474.42} C_VEL
LIN {X 0,Y 512.199,Z 282.933,A -85,B 0,C 180,E1 -5474.669,E2 -5474.669} C_VEL
LIN {X 0,Y 511.67,Z 378.479,A -85,B 0,C 180,E1 -5476.041,E2 -5476.041} C_VEL
LIN {X 0,Y 511.417,Z 392.278,A -85,B 0,C 180,E1 -5476.414,E2 -5476.414} C_VEL
LIN {X 0,Y 511.096,Z 405.167,A -85,B 0,C 180,E1 -5476.937,E2 -5476.937} C_VEL
LIN {X 0,Y 510.829,Z 416.917,A -85,B 0,C 180,E1 -5477.586,E2 -5477.586} C_VEL
LIN {X 0,Y 510.54,Z 428.272,A -85,B 0,C 180,E1 -5478.386,E2 -5478.386} C_VEL
LIN {X 0,Y 510.175,Z 438.497,A -85,B 0,C 180,E1 -5479.282,E2 -5479.282} C_VEL
LIN {X 0,Y 509.864,Z 447.69,A -85,B 0,C 180,E1 -5480.279,E2 -5480.279} C_VEL
LIN {X 0,Y 509.618,Z 456.646,A -85,B 0,C 180,E1 -5481.475,E2 -5481.475} C_VEL
LIN {X 0,Y 509.428,Z 463.854,A -85,B 0,C 180,E1 -5482.669,E2 -5482.669} C_VEL
LIN {X 0,Y 509.308,Z 468.717,A -85,B 0,C 180,E1 -5483.662,E2 -5483.662} C_VEL
LIN {X 0,Y 509.243,Z 473.444,A -85,B 0,C 180,E1 -5484.853,E2 -5484.853} C_VEL
LIN {X 0,Y 509.245,Z 477.056,A -85,B 0,C 180,E1 -5486.043,E2 -5486.043} C_VEL
LIN {X 0,Y 509.2,Z 478.918,A -85,B 0,C 180,E1 -5486.835,E2 -5486.835} C_VEL
LIN {X 0,Y 509.19,Z 480.314,A -85,B 0,C 180,E1 -5487.627,E2 -5487.627} C_VEL
LIN {X 0,Y 509.074,Z 481.913,A -85,B 0,C 180,E1 -5489.209,E2 -5489.209} C_VEL
LIN {X 0,Y 509.068,Z 482.128,A -85,B 0,C 180,E1 -5490,E2 -5490} C_VEL
LIN {X 0,Y 509.112,Z 481.303,A -85,B 0,C 180,E1 -5491.582,E2 -5491.582} C_VEL
LIN {X 0,Y 509.19,Z 480.307,A -85,B 0,C 180,E1 -5492.373,E2 -5492.373} C_VEL
LIN {X 0,Y 509.2,Z 478.908,A -85,B 0,C 180,E1 -5493.165,E2 -5493.165} C_VEL
LIN {X 0,Y 509.203,Z 475.966,A -85,B 0,C 180,E1 -5494.354,E2 -5494.354} C_VEL
LIN {X 0,Y 509.291,Z 471.986,A -85,B 0,C 180,E1 -5495.543,E2 -5495.543} C_VEL
LIN {X 0,Y 509.4,Z 465.965,A -85,B 0,C 180,E1 -5496.914,E2 -5496.914} C_VEL
LIN {X 0,Y 509.545,Z 459.171,A -85,B 0,C 180,E1 -5498.127,E2 -5498.127} C_VEL
LIN {X 0,Y 509.748,Z 450.868,A -85,B 0,C 180,E1 -5499.323,E2 -5499.323} C_VEL
LIN {X 0,Y 510.008,Z 442.355,A -85,B 0,C 180,E1 -5500.32,E2 -5500.32} C_VEL
LIN {X 0,Y 510.382,Z 431.836,A -85,B 0,C 180,E1 -5501.316,E2 -5501.316} C_VEL
LIN {X 0,Y 510.655,Z 420.838,A -85,B 0,C 180,E1 -5502.157,E2 -5502.157} C_VEL
LIN {X 0,Y 510.991,Z 410.008,A -85,B 0,C 180,E1 -5502.814,E2 -5502.814} C_VEL
LIN {X 0,Y 511.3,Z 398.253,A -85,B 0,C 180,E1 -5503.362,E2 -5503.362} C_VEL
LIN {X 0,Y 511.574,Z 385.62,A -85,B 0,C 180,E1 -5503.784,E2 -5503.784} C_VEL
LIN {X 0,Y 511.774,Z 372.722,A -85,B 0,C 180,E1 -5504.058,E2 -5504.058} C_VEL
LIN {X 0,Y 512.105,Z 281.345,A -85,B 0,C 180,E1 -5505.355,E2 -5505.355} C_VEL
LIN {X 0,Y 510.23,Z 269.441,A -85,B 0,C 180,E1 -5505.59,E2 -5505.59} C_VEL
LIN {X 0,Y 510.725,Z 249.027,A -85,B 0,C 180,E1 -5508.867,E2 -5508.867} C_VEL
LIN {X 0,Y 511.176,Z 232.354,A -85,B 0,C 180,E1 -5511.579,E2 -5511.579} C_VEL
LIN {X 0,Y 511.323,Z 224.081,A -85,B 0,C 180,E1 -5512.942,E2 -5512.942} C_VEL
LIN {X 0,Y 509.848,Z 215.977,A -85,B 0,C 180,E1 -5514.373,E2 -5514.373} C_VEL
LIN {X 0,Y 509.873,Z 215.976,A -85,B 0,C 180,E1 -5517.056,E2 -5517.056} C_VEL
LIN {X 0,Y 509.858,Z 215.975,A -85,B 0,C 180,E1 -5519.751,E2 -5519.751} C_VEL
LIN {X 0,Y 509.874,Z 215.972,A -85,B 0,C 180,E1 -5522.774,E2 -5522.774} C_VEL
LIN {X 0,Y 509.824,Z 215.981,A -85,B 0,C 180,E1 -5525.578,E2 -5525.578} C_VEL
LIN {X 0,Y 509.849,Z 215.971,A -85,B 0,C 180,E1 -5528.338,E2 -5528.338} C_VEL
LIN {X 0,Y 509.856,Z 215.977,A -85,B 0,C 180,E1 -5531.425,E2 -5531.425} C_VEL
LIN {X 0,Y 509.857,Z 215.973,A -85,B 0,C 180,E1 -5534.668,E2 -5534.668} C_VEL
LIN {X 0,Y 509.855,Z 215.969,A -85,B 0,C 180,E1 -5538.103,E2 -5538.103} C_VEL
LIN {X 0,Y 509.846,Z 215.974,A -85,B 0,C 180,E1 -5540.647,E2 -5540.647} C_VEL
LIN {X 0,Y 509.834,Z 215.975,A -85,B 0,C 180,E1 -5543.647,E2 -5543.647} C_VEL
LIN {X 0,Y 509.86,Z 215.971,A -85,B 0,C 180,E1 -5546.539,E2 -5546.539} C_VEL
LIN {X 0,Y 509.845,Z 215.977,A -85,B 0,C 180,E1 -5549.334,E2 -5549.334} C_VEL
LIN {X 0,Y 509.892,Z 215.964,A -85,B 0,C 180,E1 -5552.054,E2 -5552.054} C_VEL
LIN {X 0,Y 509.875,Z 215.971,A -85,B 0,C 180,E1 -5554.704,E2 -5554.704} C_VEL
LIN {X 0,Y 509.826,Z 215.977,A -85,B 0,C 180,E1 -5557.458,E2 -5557.458} C_VEL
LIN {X 0,Y 509.916,Z 215.963,A -85,B 0,C 180,E1 -5559.845,E2 -5559.845} C_VEL
LIN {X 0,Y 509.881,Z 215.973,A -85,B 0,C 180,E1 -5563.175,E2 -5563.175} C_VEL
LIN {X 0,Y 509.863,Z 215.967,A -85,B 0,C 180,E1 -5565.634,E2 -5565.634} C_VEL
LIN {X 0,Y 509.901,Z 215.965,A -85,B 0,C 180,E1 -5568.123,E2 -5568.123} C_VEL
LIN {X 0,Y 509.914,Z 215.966,A -85,B 0,C 180,E1 -5571.28,E2 -5571.28} C_VEL
LIN {X 0,Y 509.953,Z 215.958,A -85,B 0,C 180,E1 -5573.67,E2 -5573.67} C_VEL
LIN {X 0,Y 509.955,Z 215.966,A -85,B 0,C 180,E1 -5576.84,E2 -5576.84} C_VEL
LIN {X 0,Y 510.062,Z 215.945,A -85,B 0,C 180,E1 -5579.211,E2 -5579.211} C_VEL
LIN {X 0,Y 510.055,Z 215.949,A -85,B 0,C 180,E1 -5582.369,E2 -5582.369} C_VEL
LIN {X 0,Y 509.978,Z 215.956,A -85,B 0,C 180,E1 -5585.536,E2 -5585.536} C_VEL
LIN {X 0,Y 509.951,Z 215.957,A -85,B 0,C 180,E1 -5587.922,E2 -5587.922} C_VEL
LIN {X 0,Y 509.912,Z 215.965,A -85,B 0,C 180,E1 -5591.126,E2 -5591.126} C_VEL
LIN {X 0,Y 509.872,Z 215.973,A -85,B 0,C 180,E1 -5594.366,E2 -5594.366} C_VEL
LIN {X 0,Y 509.893,Z 215.966,A -85,B 0,C 180,E1 -5597.652,E2 -5597.652} C_VEL
LIN {X 0,Y 509.886,Z 215.973,A -85,B 0,C 180,E1 -5600.402,E2 -5600.402} C_VEL
LIN {X 0,Y 509.828,Z 215.974,A -85,B 0,C 180,E1 -5603.564,E2 -5603.564} C_VEL
LIN {X 0,Y 509.878,Z 215.974,A -85,B 0,C 180,E1 -5606.371,E2 -5606.371} C_VEL
LIN {X 0,Y 509.857,Z 215.969,A -85,B 0,C 180,E1 -5609.751,E2 -5609.751} C_VEL
LIN {X 0,Y 509.866,Z 215.977,A -85,B 0,C 180,E1 -5612.773,E2 -5612.773} C_VEL
LIN {X 0,Y 509.82,Z 215.977,A -85,B 0,C 180,E1 -5615.578,E2 -5615.578} C_VEL
LIN {X 0,Y 509.817,Z 215.984,A -85,B 0,C 180,E1 -5618.341,E2 -5618.341} C_VEL
LIN {X 0,Y 509.832,Z 215.976,A -85,B 0,C 180,E1 -5621.428,E2 -5621.428} C_VEL
LIN {X 0,Y 509.925,Z 216.132,A -85,B 0,C 180,E1 -5624.53,E2 -5624.53} C_VEL
LIN {X 0,Y 510.591,Z 220.859,A -85,B 0,C 180,E1 -5625.414,E2 -5625.414} C_VEL
LIN {X 0,Y 510.306,Z 235.346,A -85,B 0,C 180,E1 -5628.047,E2 -5628.047} C_VEL
LIN {X 0,Y 510.261,Z 243.309,A -85,B 0,C 180,E1 -5629.476,E2 -5629.476} C_VEL
LIN {X 0,Y 512.271,Z 255.276,A -85,B 0,C 180,E1 -5629.712,E2 -5629.712} C_VEL
LIN {X 0,Y 512.279,Z 264.548,A -85,B 0,C 180,E1 -5629.845,E2 -5629.845} C_VEL
LIN {X 0,Y 511.605,Z 270.388,A -85,B 0,C 180,E1 -5629.909,E2 -5629.909} C_VEL
LIN {X 0,Y 505.908,Z 289.37,A -85,B 0,C 180,E1 -5630.007,E2 -5630.007} C_VEL
LIN {X 0,Y 505.176,Z 295.212,A -85,B 0,C 180,E1 -5630.069,E2 -5630.069} C_VEL
LIN {X 0,Y 504.793,Z 351.529,A -85,B 0,C 180,E1 -5630.902,E2 -5630.902} C_VEL
LIN {X 0,Y 504.59,Z 365.075,A -85,B 0,C 180,E1 -5631.279,E2 -5631.279} C_VEL
LIN {X 0,Y 504.387,Z 377.795,A -85,B 0,C 180,E1 -5631.807,E2 -5631.807} C_VEL
LIN {X 0,Y 504.011,Z 389.251,A -85,B 0,C 180,E1 -5632.446,E2 -5632.446} C_VEL
LIN {X 0,Y 503.643,Z 400.547,A -85,B 0,C 180,E1 -5633.253,E2 -5633.253} C_VEL
LIN {X 0,Y 503.286,Z 410.728,A -85,B 0,C 180,E1 -5634.159,E2 -5634.159} C_VEL
LIN {X 0,Y 502.98,Z 420.064,A -85,B 0,C 180,E1 -5635.191,E2 -5635.191} C_VEL
LIN {X 0,Y 502.698,Z 427.855,A -85,B 0,C 180,E1 -5636.239,E2 -5636.239} C_VEL
LIN {X 0,Y 502.496,Z 435.274,A -85,B 0,C 180,E1 -5637.466,E2 -5637.466} C_VEL
LIN {X 0,Y 502.324,Z 441.781,A -85,B 0,C 180,E1 -5638.824,E2 -5638.824} C_VEL
LIN {X 0,Y 502.193,Z 446.741,A -85,B 0,C 180,E1 -5640.189,E2 -5640.189} C_VEL
LIN {X 0,Y 502.085,Z 450.421,A -85,B 0,C 180,E1 -5641.581,E2 -5641.581} C_VEL
LIN {X 0,Y 502.007,Z 452.139,A -85,B 0,C 180,E1 -5642.484,E2 -5642.484} C_VEL
LIN {X 0,Y 501.993,Z 453.533,A -85,B 0,C 180,E1 -5643.639,E2 -5643.639} C_VEL
LIN {X 0,Y 501.979,Z 454.129,A -85,B 0,C 180,E1 -5645.164,E2 -5645.164} C_VEL
LIN {X 0,Y 501.965,Z 453.812,A -85,B 0,C 180,E1 -5646.044,E2 -5646.044} C_VEL
LIN {X 0,Y 502.008,Z 452.249,A -85,B 0,C 180,E1 -5647.517,E2 -5647.517} C_VEL
LIN {X 0,Y 502.14,Z 449.026,A -85,B 0,C 180,E1 -5649.09,E2 -5649.09} C_VEL
LIN {X 0,Y 502.268,Z 445.132,A -85,B 0,C 180,E1 -5650.378,E2 -5650.378} C_VEL
LIN {X 0,Y 502.364,Z 439.851,A -85,B 0,C 180,E1 -5651.695,E2 -5651.695} C_VEL
LIN {X 0,Y 502.503,Z 433.606,A -85,B 0,C 180,E1 -5652.92,E2 -5652.92} C_VEL
LIN {X 0,Y 502.757,Z 426.982,A -85,B 0,C 180,E1 -5653.973,E2 -5653.973} C_VEL
LIN {X 0,Y 503.026,Z 418.927,A -85,B 0,C 180,E1 -5655.033,E2 -5655.033} C_VEL
LIN {X 0,Y 503.3,Z 409.303,A -85,B 0,C 180,E1 -5656.062,E2 -5656.062} C_VEL
LIN {X 0,Y 503.696,Z 398.44,A -85,B 0,C 180,E1 -5656.998,E2 -5656.998} C_VEL
LIN {X 0,Y 504.058,Z 387.945,A -85,B 0,C 180,E1 -5657.722,E2 -5657.722} C_VEL
LIN {X 0,Y 504.368,Z 376.492,A -85,B 0,C 180,E1 -5658.343,E2 -5658.343} C_VEL
LIN {X 0,Y 504.588,Z 363.647,A -85,B 0,C 180,E1 -5658.857,E2 -5658.857} C_VEL
LIN {X 0,Y 504.824,Z 350.05,A -85,B 0,C 180,E1 -5659.218,E2 -5659.218} C_VEL
LIN {X 0,Y 505.343,Z 254.729,A -85,B 0,C 180,E1 -5660.602,E2 -5660.602} C_VEL
LIN {X 0,Y 503.28,Z 243.467,A -85,B 0,C 180,E1 -5660.835,E2 -5660.835} C_VEL
LIN {X 0,Y 503.645,Z 227.04,A -85,B 0,C 180,E1 -5663.993,E2 -5663.993} C_VEL
LIN {X 0,Y 503.511,Z 220.887,A -85,B 0,C 180,E1 -5665.196,E2 -5665.196} C_VEL
LIN {X 0,Y 502.775,Z 216.861,A -85,B 0,C 180,E1 -5666.042,E2 -5666.042} C_VEL
LIN {X 0,Y 503.013,Z 216.831,A -85,B 0,C 180,E1 -5667.598,E2 -5667.598} C_VEL
LIN {X 0,Y 503.006,Z 216.829,A -85,B 0,C 180,E1 -5670,E2 -5670} C_VEL
LIN {X 0,Y 503.013,Z 216.823,A -85,B 0,C 180,E1 -5672.402,E2 -5672.402} C_VEL
LIN {X 0,Y 502.901,Z 216.845,A -85,B 0,C 180,E1 -5675.614,E2 -5675.614} C_VEL
LIN {X 0,Y 502.875,Z 216.843,A -85,B 0,C 180,E1 -5678.034,E2 -5678.034} C_VEL
LIN {X 0,Y 502.879,Z 216.844,A -85,B 0,C 180,E1 -5681.283,E2 -5681.283} C_VEL
LIN {X 0,Y 502.834,Z 216.846,A -85,B 0,C 180,E1 -5684.571,E2 -5684.571} C_VEL
LIN {X 0,Y 502.804,Z 216.853,A -85,B 0,C 180,E1 -5687.909,E2 -5687.909} C_VEL
LIN {X 0,Y 502.832,Z 216.846,A -85,B 0,C 180,E1 -5690.536,E2 -5690.536} C_VEL
LIN {X 0,Y 502.789,Z 216.854,A -85,B 0,C 180,E1 -5693.04,E2 -5693.04} C_VEL
LIN {X 0,Y 502.845,Z 216.845,A -85,B 0,C 180,E1 -5696.556,E2 -5696.556} C_VEL
LIN {X 0,Y 502.815,Z 216.851,A -85,B 0,C 180,E1 -5699.934,E2 -5699.934} C_VEL
LIN {X 0,Y 502.833,Z 216.85,A -85,B 0,C 180,E1 -5703.031,E2 -5703.031} C_VEL
LIN {X 0,Y 502.768,Z 216.857,A -85,B 0,C 180,E1 -5705.951,E2 -5705.951} C_VEL
LIN {X 0,Y 502.801,Z 216.854,A -85,B 0,C 180,E1 -5708.976,E2 -5708.976} C_VEL
LIN {X 0,Y 502.803,Z 216.851,A -85,B 0,C 180,E1 -5712.199,E2 -5712.199} C_VEL
LIN {X 0,Y 502.785,Z 216.859,A -85,B 0,C 180,E1 -5715.47,E2 -5715.47} C_VEL
LIN {X 0,Y 502.818,Z 216.852,A -85,B 0,C 180,E1 -5718.934,E2 -5718.934} C_VEL
LIN {X 0,Y 502.792,Z 216.853,A -85,B 0,C 180,E1 -5722.046,E2 -5722.046} C_VEL
LIN {X 0,Y 502.806,Z 216.854,A -85,B 0,C 180,E1 -5725.034,E2 -5725.034} C_VEL
LIN {X 0,Y 502.781,Z 216.855,A -85,B 0,C 180,E1 -5727.915,E2 -5727.915} C_VEL
LIN {X 0,Y 502.822,Z 216.851,A -85,B 0,C 180,E1 -5730.712,E2 -5730.712} C_VEL
LIN {X 0,Y 502.861,Z 216.849,A -85,B 0,C 180,E1 -5733.439,E2 -5733.439} C_VEL
LIN {X 0,Y 502.79,Z 216.853,A -85,B 0,C 180,E1 -5736.086,E2 -5736.086} C_VEL
LIN {X 0,Y 502.781,Z 216.856,A -85,B 0,C 180,E1 -5738.689,E2 -5738.689} C_VEL
LIN {X 0,Y 502.827,Z 216.852,A -85,B 0,C 180,E1 -5741.248,E2 -5741.248} C_VEL
LIN {X 0,Y 502.819,Z 216.85,A -85,B 0,C 180,E1 -5743.767,E2 -5743.767} C_VEL
LIN {X 0,Y 502.828,Z 216.848,A -85,B 0,C 180,E1 -5746.254,E2 -5746.254} C_VEL
LIN {X 0,Y 502.875,Z 216.846,A -85,B 0,C 180,E1 -5748.717,E2 -5748.717} C_VEL
LIN {X 0,Y 502.899,Z 216.839,A -85,B 0,C 180,E1 -5751.967,E2 -5751.967} C_VEL
LIN {X 0,Y 502.938,Z 216.835,A -85,B 0,C 180,E1 -5754.386,E2 -5754.386} C_VEL
LIN {X 0,Y 503.023,Z 216.825,A -85,B 0,C 180,E1 -5757.598,E2 -5757.598} C_VEL
LIN {X 0,Y 503.025,Z 216.823,A -85,B 0,C 180,E1 -5760,E2 -5760} C_VEL
LIN {X 0,Y 503.023,Z 216.825,A -85,B 0,C 180,E1 -5762.402,E2 -5762.402} C_VEL
LIN {X 0,Y 502.939,Z 216.835,A -85,B 0,C 180,E1 -5765.613,E2 -5765.613} C_VEL
LIN {X 0,Y 502.899,Z 216.839,A -85,B 0,C 180,E1 -5768.033,E2 -5768.033} C_VEL
LIN {X 0,Y 502.874,Z 216.846,A -85,B 0,C 180,E1 -5771.283,E2 -5771.283} C_VEL
LIN {X 0,Y 502.842,Z 216.85,A -85,B 0,C 180,E1 -5774.571,E2 -5774.571} C_VEL
LIN {X 0,Y 502.859,Z 216.844,A -85,B 0,C 180,E1 -5777.907,E2 -5777.907} C_VEL
LIN {X 0,Y 502.826,Z 216.852,A -85,B 0,C 180,E1 -5780.536,E2 -5780.536} C_VEL
LIN {X 0,Y 502.795,Z 216.855,A -85,B 0,C 180,E1 -5783.04,E2 -5783.04} C_VEL
LIN {X 0,Y 502.838,Z 216.846,A -85,B 0,C 180,E1 -5785.676,E2 -5785.676} C_VEL
LIN {X 0,Y 502.837,Z 216.849,A -85,B 0,C 180,E1 -5788.373,E2 -5788.373} C_VEL
LIN {X 0,Y 502.79,Z 216.853,A -85,B 0,C 180,E1 -5791.499,E2 -5791.499} C_VEL
LIN {X 0,Y 502.803,Z 216.855,A -85,B 0,C 180,E1 -5794.445,E2 -5794.445} C_VEL
LIN {X 0,Y 502.778,Z 216.856,A -85,B 0,C 180,E1 -5797.179,E2 -5797.179} C_VEL
LIN {X 0,Y 502.786,Z 216.853,A -85,B 0,C 180,E1 -5800.016,E2 -5800.016} C_VEL
LIN {X 0,Y 502.801,Z 216.852,A -85,B 0,C 180,E1 -5802.2,E2 -5802.2} C_VEL
LIN {X 0,Y 502.8,Z 216.851,A -85,B 0,C 180,E1 -5805.469,E2 -5805.469} C_VEL
LIN {X 0,Y 502.819,Z 216.851,A -85,B 0,C 180,E1 -5808.934,E2 -5808.934} C_VEL
LIN {X 0,Y 502.789,Z 216.853,A -85,B 0,C 180,E1 -5812.046,E2 -5812.046} C_VEL
LIN {X 0,Y 502.797,Z 216.853,A -85,B 0,C 180,E1 -5815.034,E2 -5815.034} C_VEL
LIN {X 0,Y 502.784,Z 216.852,A -85,B 0,C 180,E1 -5817.916,E2 -5817.916} C_VEL
LIN {X 0,Y 502.822,Z 216.855,A -85,B 0,C 180,E1 -5820.712,E2 -5820.712} C_VEL
LIN {X 0,Y 502.845,Z 216.849,A -85,B 0,C 180,E1 -5823.444,E2 -5823.444} C_VEL
LIN {X 0,Y 502.806,Z 216.956,A -85,B 0,C 180,E1 -5825.344,E2 -5825.344} C_VEL
LIN {X 0,Y 504.516,Z 226.384,A -85,B 0,C 180,E1 -5827.043,E2 -5827.043} C_VEL
LIN {X 0,Y 504.004,Z 242.876,A -85,B 0,C 180,E1 -5829.811,E2 -5829.811} C_VEL
LIN {X 0,Y 503.488,Z 260.619,A -85,B 0,C 180,E1 -5832.746,E2 -5832.746} C_VEL
LIN {X 0,Y 503.26,Z 269.604,A -85,B 0,C 180,E1 -5834.199,E2 -5834.199} C_VEL
LIN {X 0,Y 505.34,Z 283.146,A -85,B 0,C 180,E1 -5834.462,E2 -5834.462} C_VEL
LIN {X 0,Y 504.777,Z 378.218,A -85,B 0,C 180,E1 -5835.847,E2 -5835.847} C_VEL
LIN {X 0,Y 504.498,Z 392.038,A -85,B 0,C 180,E1 -5836.224,E2 -5836.224} C_VEL
LIN {X 0,Y 504.175,Z 404.944,A -85,B 0,C 180,E1 -5836.754,E2 -5836.754} C_VEL
LIN {X 0,Y 503.884,Z 416.323,A -85,B 0,C 180,E1 -5837.388,E2 -5837.388} C_VEL
LIN {X 0,Y 503.588,Z 426.763,A -85,B 0,C 180,E1 -5838.121,E2 -5838.121} C_VEL
LIN {X 0,Y 503.233,Z 437.237,A -85,B 0,C 180,E1 -5839.031,E2 -5839.031} C_VEL
LIN {X 0,Y 502.892,Z 445.798,A -85,B 0,C 180,E1 -5839.94,E2 -5839.94} C_VEL
LIN {X 0,Y 502.637,Z 453.697,A -85,B 0,C 180,E1 -5840.95,E2 -5840.95} C_VEL
LIN {X 0,Y 502.397,Z 461.411,A -85,B 0,C 180,E1 -5842.161,E2 -5842.161} C_VEL
LIN {X 0,Y 502.235,Z 468.518,A -85,B 0,C 180,E1 -5843.573,E2 -5843.573} C_VEL
LIN {X 0,Y 502.174,Z 473.247,A -85,B 0,C 180,E1 -5844.781,E2 -5844.781} C_VEL
LIN {X 0,Y 502.138,Z 476.859,A -85,B 0,C 180,E1 -5845.987,E2 -5845.987} C_VEL
LIN {X 0,Y 502.12,Z 478.722,A -85,B 0,C 180,E1 -5846.791,E2 -5846.791} C_VEL
LIN {X 0,Y 502.091,Z 480.118,A -85,B 0,C 180,E1 -5847.593,E2 -5847.593} C_VEL
LIN {X 0,Y 501.991,Z 481.718,A -85,B 0,C 180,E1 -5849.198,E2 -5849.198} C_VEL
LIN {X 0,Y 501.982,Z 481.932,A -85,B 0,C 180,E1 -5850,E2 -5850} C_VEL
LIN {X 0,Y 502.036,Z 481.105,A -85,B 0,C 180,E1 -5851.604,E2 -5851.604} C_VEL
LIN {X 0,Y 502.092,Z 480.108,A -85,B 0,C 180,E1 -5852.407,E2 -5852.407} C_VEL
LIN {X 0,Y 502.12,Z 478.709,A -85,B 0,C 180,E1 -5853.21,E2 -5853.21} C_VEL
LIN {X 0,Y 502.101,Z 475.764,A -85,B 0,C 180,E1 -5854.415,E2 -5854.415} C_VEL
LIN {X 0,Y 502.207,Z 471.783,A -85,B 0,C 180,E1 -5855.622,E2 -5855.622} C_VEL
LIN {X 0,Y 502.33,Z 465.758,A -85,B 0,C 180,E1 -5857.012,E2 -5857.012} C_VEL
LIN {X 0,Y 502.478,Z 458.961,A -85,B 0,C 180,E1 -5858.243,E2 -5858.243} C_VEL
LIN {X 0,Y 502.717,Z 450.656,A -85,B 0,C 180,E1 -5859.455,E2 -5859.455} C_VEL
LIN {X 0,Y 502.99,Z 442.137,A -85,B 0,C 180,E1 -5860.465,E2 -5860.465} C_VEL
LIN {X 0,Y 503.402,Z 431.614,A -85,B 0,C 180,E1 -5861.475,E2 -5861.475} C_VEL
LIN {X 0,Y 503.696,Z 420.61,A -85,B 0,C 180,E1 -5862.327,E2 -5862.327} C_VEL
LIN {X 0,Y 504.046,Z 409.775,A -85,B 0,C 180,E1 -5862.993,E2 -5862.993} C_VEL
LIN {X 0,Y 504.378,Z 398.009,A -85,B 0,C 180,E1 -5863.548,E2 -5863.548} C_VEL
LIN {X 0,Y 504.661,Z 384.447,A -85,B 0,C 180,E1 -5864.003,E2 -5864.003} C_VEL
LIN {X 0,Y 504.902,Z 370.81,A -85,B 0,C 180,E1 -5864.279,E2 -5864.279} C_VEL
LIN {X 0,Y 505.227,Z 281.837,A -85,B 0,C 180,E1 -5865.559,E2 -5865.559} C_VEL
LIN {X 0,Y 503.219,Z 269.192,A -85,B 0,C 180,E1 -5865.82,E2 -5865.82} C_VEL
LIN {X 0,Y 503.741,Z 250.097,A -85,B 0,C 180,E1 -5868.928,E2 -5868.928} C_VEL
LIN {X 0,Y 504.225,Z 233.432,A -85,B 0,C 180,E1 -5871.676,E2 -5871.676} C_VEL
LIN {X 0,Y 504.313,Z 224.879,A -85,B 0,C 180,E1 -5873.108,E2 -5873.108} C_VEL
LIN {X 0,Y 502.794,Z 216.857,A -85,B 0,C 180,E1 -5874.561,E2 -5874.561} C_VEL
LIN {X 0,Y 502.824,Z 216.854,A -85,B 0,C 180,E1 -5877.467,E2 -5877.467} C_VEL
LIN {X 0,Y 502.809,Z 216.85,A -85,B 0,C 180,E1 -5880.211,E2 -5880.211} C_VEL
LIN {X 0,Y 502.833,Z 216.852,A -85,B 0,C 180,E1 -5883.031,E2 -5883.031} C_VEL
LIN {X 0,Y 502.768,Z 216.856,A -85,B 0,C 180,E1 -5885.951,E2 -5885.951} C_VEL
LIN {X 0,Y 502.801,Z 216.854,A -85,B 0,C 180,E1 -5888.976,E2 -5888.976} C_VEL
LIN {X 0,Y 502.796,Z 216.85,A -85,B 0,C 180,E1 -5892.139,E2 -5892.139} C_VEL
LIN {X 0,Y 502.801,Z 216.856,A -85,B 0,C 180,E1 -5895.468,E2 -5895.468} C_VEL
LIN {X 0,Y 502.819,Z 216.85,A -85,B 0,C 180,E1 -5898.934,E2 -5898.934} C_VEL
LIN {X 0,Y 502.793,Z 216.85,A -85,B 0,C 180,E1 -5902.046,E2 -5902.046} C_VEL
LIN {X 0,Y 502.807,Z 216.854,A -85,B 0,C 180,E1 -5905.035,E2 -5905.035} C_VEL
LIN {X 0,Y 502.782,Z 216.85,A -85,B 0,C 180,E1 -5907.915,E2 -5907.915} C_VEL
LIN {X 0,Y 502.824,Z 216.85,A -85,B 0,C 180,E1 -5910.712,E2 -5910.712} C_VEL
LIN {X 0,Y 502.862,Z 216.845,A -85,B 0,C 180,E1 -5913.439,E2 -5913.439} C_VEL
LIN {X 0,Y 502.785,Z 216.85,A -85,B 0,C 180,E1 -5916.086,E2 -5916.086} C_VEL
LIN {X 0,Y 502.782,Z 216.855,A -85,B 0,C 180,E1 -5918.689,E2 -5918.689} C_VEL
LIN {X 0,Y 502.828,Z 216.849,A -85,B 0,C 180,E1 -5921.248,E2 -5921.248} C_VEL
LIN {X 0,Y 502.82,Z 216.847,A -85,B 0,C 180,E1 -5923.767,E2 -5923.767} C_VEL
LIN {X 0,Y 502.834,Z 216.842,A -85,B 0,C 180,E1 -5926.255,E2 -5926.255} C_VEL
LIN {X 0,Y 502.876,Z 216.845,A -85,B 0,C 180,E1 -5928.717,E2 -5928.717} C_VEL
LIN {X 0,Y 502.901,Z 216.836,A -85,B 0,C 180,E1 -5931.967,E2 -5931.967} C_VEL
LIN {X 0,Y 502.932,Z 216.834,A -85,B 0,C 180,E1 -5934.386,E2 -5934.386} C_VEL
LIN {X 0,Y 503.024,Z 216.822,A -85,B 0,C 180,E1 -5937.598,E2 -5937.598} C_VEL
LIN {X 0,Y 503.027,Z 216.818,A -85,B 0,C 180,E1 -5940,E2 -5940} C_VEL
LIN {X 0,Y 503.024,Z 216.825,A -85,B 0,C 180,E1 -5942.402,E2 -5942.402} C_VEL
LIN {X 0,Y 502.932,Z 216.833,A -85,B 0,C 180,E1 -5945.614,E2 -5945.614} C_VEL
LIN {X 0,Y 502.901,Z 216.835,A -85,B 0,C 180,E1 -5948.033,E2 -5948.033} C_VEL
LIN {X 0,Y 502.876,Z 216.839,A -85,B 0,C 180,E1 -5951.283,E2 -5951.283} C_VEL
LIN {X 0,Y 502.851,Z 216.851,A -85,B 0,C 180,E1 -5954.571,E2 -5954.571} C_VEL
LIN {X 0,Y 502.855,Z 216.843,A -85,B 0,C 180,E1 -5957.907,E2 -5957.907} C_VEL
LIN {X 0,Y 502.828,Z 216.854,A -85,B 0,C 180,E1 -5960.536,E2 -5960.536} C_VEL
LIN {X 0,Y 502.79,Z 216.853,A -85,B 0,C 180,E1 -5963.041,E2 -5963.041} C_VEL
LIN {X 0,Y 502.798,Z 216.85,A -85,B 0,C 180,E1 -5965.678,E2 -5965.678} C_VEL
LIN {X 0,Y 502.796,Z 216.857,A -85,B 0,C 180,E1 -5968.376,E2 -5968.376} C_VEL
LIN {X 0,Y 502.795,Z 216.852,A -85,B 0,C 180,E1 -5971.144,E2 -5971.144} C_VEL
LIN {X 0,Y 502.788,Z 216.856,A -85,B 0,C 180,E1 -5973.995,E2 -5973.995} C_VEL
LIN {X 0,Y 502.753,Z 216.858,A -85,B 0,C 180,E1 -5977.174,E2 -5977.174} C_VEL
LIN {X 0,Y 502.771,Z 216.858,A -85,B 0,C 180,E1 -5980.017,E2 -5980.017} C_VEL
LIN {X 0,Y 502.771,Z 216.86,A -85,B 0,C 180,E1 -5982.195,E2 -5982.195} C_VEL
LIN {X 0,Y 502.883,Z 217.041,A -85,B 0,C 180,E1 -5984.398,E2 -5984.398} C_VEL
LIN {X 0,Y 503.628,Z 222.167,A -85,B 0,C 180,E1 -5985.373,E2 -5985.373} C_VEL
LIN {X 0,Y 503.307,Z 237.521,A -85,B 0,C 180,E1 -5988.183,E2 -5988.183} C_VEL
LIN {X 0,Y 503.287,Z 243.46,A -85,B 0,C 180,E1 -5989.253,E2 -5989.253} C_VEL
LIN {X 0,Y 505.443,Z 255.818,A -85,B 0,C 180,E1 -5989.505,E2 -5989.505} C_VEL
LIN {X 0,Y 505.176,Z 295.212,A -85,B 0,C 180,E1 -5990.069,E2 -5990.069} C_VEL
LIN {X 0,Y 504.451,Z 301.056,A -85,B 0,C 180,E1 -5990.132,E2 -5990.132} C_VEL
LIN {X 0,Y 498.812,Z 320.052,A -85,B 0,C 180,E1 -5990.237,E2 -5990.237} C_VEL
LIN {X 0,Y 498.143,Z 325.893,A -85,B 0,C 180,E1 -5990.303,E2 -5990.303} C_VEL
LIN {X 0,Y 497.911,Z 352.305,A -85,B 0,C 180,E1 -5990.717,E2 -5990.717} C_VEL
LIN {X 0,Y 497.707,Z 365.325,A -85,B 0,C 180,E1 -5991.087,E2 -5991.087} C_VEL
LIN {X 0,Y 497.477,Z 378.056,A -85,B 0,C 180,E1 -5991.624,E2 -5991.624} C_VEL
LIN {X 0,Y 497.079,Z 389.71,A -85,B 0,C 180,E1 -5992.286,E2 -5992.286} C_VEL
LIN {X 0,Y 496.649,Z 401.626,A -85,B 0,C 180,E1 -5993.156,E2 -5993.156} C_VEL
LIN {X 0,Y 496.283,Z 412.378,A -85,B 0,C 180,E1 -5994.158,E2 -5994.158} C_VEL
LIN {X 0,Y 495.895,Z 422.119,A -85,B 0,C 180,E1 -5995.286,E2 -5995.286} C_VEL
LIN {X 0,Y 495.608,Z 430.087,A -85,B 0,C 180,E1 -5996.424,E2 -5996.424} C_VEL
LIN {X 0,Y 495.436,Z 436.855,A -85,B 0,C 180,E1 -5997.622,E2 -5997.622} C_VEL
LIN {X 0,Y 495.245,Z 442.308,A -85,B 0,C 180,E1 -5998.819,E2 -5998.819} C_VEL
LIN {X 0,Y 495.101,Z 447.211,A -85,B 0,C 180,E1 -6000.21,E2 -6000.21} C_VEL
LIN {X 0,Y 494.995,Z 450.936,A -85,B 0,C 180,E1 -6001.677,E2 -6001.677} C_VEL
LIN {X 0,Y 494.902,Z 453.057,A -85,B 0,C 180,E1 -6002.972,E2 -6002.972} C_VEL
LIN {X 0,Y 494.909,Z 453.928,A -85,B 0,C 180,E1 -6003.882,E2 -6003.882} C_VEL
LIN {X 0,Y 494.884,Z 454.288,A -85,B 0,C 180,E1 -6005.352,E2 -6005.352} C_VEL
LIN {X 0,Y 494.858,Z 453.625,A -85,B 0,C 180,E1 -6006.568,E2 -6006.568} C_VEL
LIN {X 0,Y 494.916,Z 452.577,A -85,B 0,C 180,E1 -6007.455,E2 -6007.455} C_VEL
LIN {X 0,Y 495.003,Z 450.123,A -85,B 0,C 180,E1 -6008.774,E2 -6008.774} C_VEL
LIN {X 0,Y 495.172,Z 446.558,A -85,B 0,C 180,E1 -6010.085,E2 -6010.085} C_VEL
LIN {X 0,Y 495.268,Z 441.834,A -85,B 0,C 180,E1 -6011.381,E2 -6011.381} C_VEL
LIN {X 0,Y 495.404,Z 435.775,A -85,B 0,C 180,E1 -6012.668,E2 -6012.668} C_VEL
LIN {X 0,Y 495.686,Z 428.161,A -85,B 0,C 180,E1 -6013.95,E2 -6013.95} C_VEL
LIN {X 0,Y 495.978,Z 420.085,A -85,B 0,C 180,E1 -6015.052,E2 -6015.052} C_VEL
LIN {X 0,Y 496.331,Z 410.977,A -85,B 0,C 180,E1 -6016.071,E2 -6016.071} C_VEL
LIN {X 0,Y 496.63,Z 401.794,A -85,B 0,C 180,E1 -6016.913,E2 -6016.913} C_VEL
LIN {X 0,Y 497.053,Z 390.361,A -85,B 0,C 180,E1 -6017.755,E2 -6017.755} C_VEL
LIN {X 0,Y 497.397,Z 378.558,A -85,B 0,C 180,E1 -6018.436,E2 -6018.436} C_VEL
LIN {X 0,Y 497.672,Z 366.523,A -85,B 0,C 180,E1 -6018.958,E2 -6018.958} C_VEL
LIN {X 0,Y 497.924,Z 353.156,A -85,B 0,C 180,E1 -6019.35,E2 -6019.35} C_VEL
LIN {X 0,Y 498.098,Z 332.528,A -85,B 0,C 180,E1 -6019.687,E2 -6019.687} C_VEL
LIN {X 0,Y 498.54,Z 255.72,A -85,B 0,C 180,E1 -6020.807,E2 -6020.807} C_VEL
LIN {X 0,Y 496.27,Z 243.63,A -85,B 0,C 180,E1 -6021.064,E2 -6021.064} C_VEL
LIN {X 0,Y 496.688,Z 227.943,A -85,B 0,C 180,E1 -6024.112,E2 -6024.112} C_VEL
LIN {X 0,Y 496.62,Z 222.791,A -85,B 0,C 180,E1 -6025.129,E2 -6025.129} C_VEL
LIN {X 0,Y 495.739,Z 217.736,A -85,B 0,C 180,E1 -6026.19,E2 -6026.19} C_VEL
LIN {X 0,Y 495.98,Z 217.707,A -85,B 0,C 180,E1 -6027.564,E2 -6027.564} C_VEL
LIN {X 0,Y 495.975,Z 217.705,A -85,B 0,C 180,E1 -6030,E2 -6030} C_VEL
LIN {X 0,Y 495.98,Z 217.699,A -85,B 0,C 180,E1 -6032.436,E2 -6032.436} C_VEL
LIN {X 0,Y 495.859,Z 217.722,A -85,B 0,C 180,E1 -6035.694,E2 -6035.694} C_VEL
LIN {X 0,Y 495.833,Z 217.719,A -85,B 0,C 180,E1 -6038.148,E2 -6038.148} C_VEL
LIN {X 0,Y 495.854,Z 217.72,A -85,B 0,C 180,E1 -6041.445,E2 -6041.445} C_VEL
LIN {X 0,Y 495.783,Z 217.725,A -85,B 0,C 180,E1 -6044.783,E2 -6044.783} C_VEL
LIN {X 0,Y 495.781,Z 217.726,A -85,B 0,C 180,E1 -6048.171,E2 -6048.171} C_VEL
LIN {X 0,Y 495.776,Z 217.726,A -85,B 0,C 180,E1 -6050.756,E2 -6050.756} C_VEL
LIN {X 0,Y 495.741,Z 217.735,A -85,B 0,C 180,E1 -6053.387,E2 -6053.387} C_VEL
LIN {X 0,Y 495.776,Z 217.726,A -85,B 0,C 180,E1 -6056.737,E2 -6056.737} C_VEL
LIN {X 0,Y 495.764,Z 217.732,A -85,B 0,C 180,E1 -6059.746,E2 -6059.746} C_VEL
LIN {X 0,Y 495.768,Z 217.727,A -85,B 0,C 180,E1 -6062.594,E2 -6062.594} C_VEL
LIN {X 0,Y 495.746,Z 217.736,A -85,B 0,C 180,E1 -6065.537,E2 -6065.537} C_VEL
LIN {X 0,Y 495.762,Z 217.729,A -85,B 0,C 180,E1 -6068.768,E2 -6068.768} C_VEL
LIN {X 0,Y 495.75,Z 217.732,A -85,B 0,C 180,E1 -6071.781,E2 -6071.781} C_VEL
LIN {X 0,Y 495.736,Z 217.734,A -85,B 0,C 180,E1 -6075.14,E2 -6075.14} C_VEL
LIN {X 0,Y 495.755,Z 217.729,A -85,B 0,C 180,E1 -6078.218,E2 -6078.218} C_VEL
LIN {X 0,Y 495.749,Z 217.735,A -85,B 0,C 180,E1 -6081.408,E2 -6081.408} C_VEL
LIN {X 0,Y 495.754,Z 217.73,A -85,B 0,C 180,E1 -6084.463,E2 -6084.463} C_VEL
LIN {X 0,Y 495.766,Z 217.732,A -85,B 0,C 180,E1 -6087.405,E2 -6087.405} C_VEL
LIN {X 0,Y 495.764,Z 217.728,A -85,B 0,C 180,E1 -6090.253,E2 -6090.253} C_VEL
LIN {X 0,Y 495.821,Z 217.725,A -85,B 0,C 180,E1 -6093.25,E2 -6093.25} C_VEL
LIN {X 0,Y 495.75,Z 217.732,A -85,B 0,C 180,E1 -6095.725,E2 -6095.725} C_VEL
LIN {X 0,Y 495.745,Z 217.731,A -85,B 0,C 180,E1 -6098.371,E2 -6098.371} C_VEL
LIN {X 0,Y 495.781,Z 217.73,A -85,B 0,C 180,E1 -6100.971,E2 -6100.971} C_VEL
LIN {X 0,Y 495.775,Z 217.73,A -85,B 0,C 180,E1 -6103.53,E2 -6103.53} C_VEL
LIN {X 0,Y 495.791,Z 217.725,A -85,B 0,C 180,E1 -6106.055,E2 -6106.055} C_VEL
LIN {X 0,Y 495.849,Z 217.72,A -85,B 0,C 180,E1 -6108.555,E2 -6108.555} C_VEL
LIN {X 0,Y 495.871,Z 217.715,A -85,B 0,C 180,E1 -6111.852,E2 -6111.852} C_VEL
LIN {X 0,Y 495.896,Z 217.712,A -85,B 0,C 180,E1 -6114.306,E2 -6114.306} C_VEL
LIN {X 0,Y 495.991,Z 217.702,A -85,B 0,C 180,E1 -6117.564,E2 -6117.564} C_VEL
LIN {X 0,Y 495.996,Z 217.699,A -85,B 0,C 180,E1 -6120,E2 -6120} C_VEL
LIN {X 0,Y 495.991,Z 217.701,A -85,B 0,C 180,E1 -6122.436,E2 -6122.436} C_VEL
LIN {X 0,Y 495.896,Z 217.712,A -85,B 0,C 180,E1 -6125.693,E2 -6125.693} C_VEL
LIN {X 0,Y 495.87,Z 217.715,A -85,B 0,C 180,E1 -6128.148,E2 -6128.148} C_VEL
LIN {X 0,Y 495.849,Z 217.719,A -85,B 0,C 180,E1 -6131.445,E2 -6131.445} C_VEL
LIN {X 0,Y 495.787,Z 217.73,A -85,B 0,C 180,E1 -6134.783,E2 -6134.783} C_VEL
LIN {X 0,Y 495.784,Z 217.728,A -85,B 0,C 180,E1 -6137.319,E2 -6137.319} C_VEL
LIN {X 0,Y 495.775,Z 217.726,A -85,B 0,C 180,E1 -6139.89,E2 -6139.89} C_VEL
LIN {X 0,Y 495.756,Z 217.733,A -85,B 0,C 180,E1 -6142.861,E2 -6142.861} C_VEL
LIN {X 0,Y 495.788,Z 217.725,A -85,B 0,C 180,E1 -6146.068,E2 -6146.068} C_VEL
LIN {X 0,Y 495.77,Z 217.732,A -85,B 0,C 180,E1 -6148.815,E2 -6148.815} C_VEL
LIN {X 0,Y 495.753,Z 217.729,A -85,B 0,C 180,E1 -6151.726,E2 -6151.726} C_VEL
LIN {X 0,Y 495.773,Z 217.732,A -85,B 0,C 180,E1 -6154.695,E2 -6154.695} C_VEL
LIN {X 0,Y 495.729,Z 217.732,A -85,B 0,C 180,E1 -6157.562,E2 -6157.562} C_VEL
LIN {X 0,Y 495.764,Z 217.733,A -85,B 0,C 180,E1 -6160.7,E2 -6160.7} C_VEL
LIN {X 0,Y 495.732,Z 217.732,A -85,B 0,C 180,E1 -6164.001,E2 -6164.001} C_VEL
LIN {X 0,Y 495.725,Z 217.734,A -85,B 0,C 180,E1 -6167.117,E2 -6167.117} C_VEL
LIN {X 0,Y 495.758,Z 217.728,A -85,B 0,C 180,E1 -6169.953,E2 -6169.953} C_VEL
LIN {X 0,Y 495.718,Z 217.74,A -85,B 0,C 180,E1 -6172.555,E2 -6172.555} C_VEL
LIN {X 0,Y 495.777,Z 217.725,A -85,B 0,C 180,E1 -6175.457,E2 -6175.457} C_VEL
LIN {X 0,Y 495.756,Z 217.733,A -85,B 0,C 180,E1 -6178.364,E2 -6178.364} C_VEL
LIN {X 0,Y 495.785,Z 217.726,A -85,B 0,C 180,E1 -6181.508,E2 -6181.508} C_VEL
LIN {X 0,Y 495.755,Z 217.734,A -85,B 0,C 180,E1 -6183.93,E2 -6183.93} C_VEL
LIN {X 0,Y 495.73,Z 217.74,A -85,B 0,C 180,E1 -6185.14,E2 -6185.14} C_VEL
LIN {X 0,Y 497.532,Z 226.937,A -85,B 0,C 180,E1 -6186.83,E2 -6186.83} C_VEL
LIN {X 0,Y 497.111,Z 241.419,A -85,B 0,C 180,E1 -6189.302,E2 -6189.302} C_VEL
LIN {X 0,Y 496.531,Z 259.162,A -85,B 0,C 180,E1 -6192.283,E2 -6192.283} C_VEL
LIN {X 0,Y 496.258,Z 269.262,A -85,B 0,C 180,E1 -6193.964,E2 -6193.964} C_VEL
LIN {X 0,Y 498.507,Z 284.064,A -85,B 0,C 180,E1 -6194.261,E2 -6194.261} C_VEL
LIN {X 0,Y 497.902,Z 377.93,A -85,B 0,C 180,E1 -6195.647,E2 -6195.647} C_VEL
LIN {X 0,Y 497.593,Z 391.781,A -85,B 0,C 180,E1 -6196.029,E2 -6196.029} C_VEL
LIN {X 0,Y 497.258,Z 404.71,A -85,B 0,C 180,E1 -6196.567,E2 -6196.567} C_VEL
LIN {X 0,Y 496.911,Z 416.539,A -85,B 0,C 180,E1 -6197.237,E2 -6197.237} C_VEL
LIN {X 0,Y 496.583,Z 427.842,A -85,B 0,C 180,E1 -6198.055,E2 -6198.055} C_VEL
LIN {X 0,Y 496.197,Z 438.079,A -85,B 0,C 180,E1 -6198.977,E2 -6198.977} C_VEL
LIN {X 0,Y 495.812,Z 447.279,A -85,B 0,C 180,E1 -6200.001,E2 -6200.001} C_VEL
LIN {X 0,Y 495.512,Z 456.24,A -85,B 0,C 180,E1 -6201.23,E2 -6201.23} C_VEL
LIN {X 0,Y 495.276,Z 463.452,A -85,B 0,C 180,E1 -6202.458,E2 -6202.458} C_VEL
LIN {X 0,Y 495.123,Z 469.511,A -85,B 0,C 180,E1 -6203.761,E2 -6203.761} C_VEL
LIN {X 0,Y 495.035,Z 474.363,A -85,B 0,C 180,E1 -6205.114,E2 -6205.114} C_VEL
LIN {X 0,Y 495.031,Z 476.661,A -85,B 0,C 180,E1 -6205.93,E2 -6205.93} C_VEL
LIN {X 0,Y 495.041,Z 478.526,A -85,B 0,C 180,E1 -6206.745,E2 -6206.745} C_VEL
LIN {X 0,Y 494.998,Z 479.922,A -85,B 0,C 180,E1 -6207.559,E2 -6207.559} C_VEL
LIN {X 0,Y 494.962,Z 480.916,A -85,B 0,C 180,E1 -6208.373,E2 -6208.373} C_VEL
LIN {X 0,Y 494.9,Z 481.736,A -85,B 0,C 180,E1 -6210,E2 -6210} C_VEL
LIN {X 0,Y 494.962,Z 480.908,A -85,B 0,C 180,E1 -6211.627,E2 -6211.627} C_VEL
LIN {X 0,Y 494.998,Z 479.91,A -85,B 0,C 180,E1 -6212.441,E2 -6212.441} C_VEL
LIN {X 0,Y 495.042,Z 478.51,A -85,B 0,C 180,E1 -6213.256,E2 -6213.256} C_VEL
LIN {X 0,Y 495.007,Z 475.563,A -85,B 0,C 180,E1 -6214.479,E2 -6214.479} C_VEL
LIN {X 0,Y 495.124,Z 471.579,A -85,B 0,C 180,E1 -6215.702,E2 -6215.702} C_VEL
LIN {X 0,Y 495.255,Z 465.449,A -85,B 0,C 180,E1 -6217.133,E2 -6217.133} C_VEL
LIN {X 0,Y 495.426,Z 458.752,A -85,B 0,C 180,E1 -6218.361,E2 -6218.361} C_VEL
LIN {X 0,Y 495.694,Z 450.444,A -85,B 0,C 180,E1 -6219.59,E2 -6219.59} C_VEL
LIN {X 0,Y 495.985,Z 441.923,A -85,B 0,C 180,E1 -6220.615,E2 -6220.615} C_VEL
LIN {X 0,Y 496.42,Z 431.396,A -85,B 0,C 180,E1 -6221.639,E2 -6221.639} C_VEL
LIN {X 0,Y 496.755,Z 420.084,A -85,B 0,C 180,E1 -6222.525,E2 -6222.525} C_VEL
LIN {X 0,Y 497.102,Z 409.549,A -85,B 0,C 180,E1 -6223.178,E2 -6223.178} C_VEL
LIN {X 0,Y 497.445,Z 397.774,A -85,B 0,C 180,E1 -6223.741,E2 -6223.741} C_VEL
LIN {X 0,Y 497.78,Z 384.203,A -85,B 0,C 180,E1 -6224.2,E2 -6224.2} C_VEL
LIN {X 0,Y 498.022,Z 370.532,A -85,B 0,C 180,E1 -6224.48,E2 -6224.48} C_VEL
LIN {X 0,Y 498.454,Z 283.182,A -85,B 0,C 180,E1 -6225.754,E2 -6225.754} C_VEL
LIN {X 0,Y 496.22,Z 269.058,A -85,B 0,C 180,E1 -6226.037,E2 -6226.037} C_VEL
LIN {X 0,Y 496.78,Z 249.895,A -85,B 0,C 180,E1 -6229.203,E2 -6229.203} C_VEL
LIN {X 0,Y 497.286,Z 234.506,A -85,B 0,C 180,E1 -6231.776,E2 -6231.776} C_VEL
LIN {X 0,Y 497.411,Z 226.472,A -85,B 0,C 180,E1 -6233.137,E2 -6233.137} C_VEL
LIN {X 0,Y 495.744,Z 217.735,A -85,B 0,C 180,E1 -6234.737,E2 -6234.737} C_VEL
LIN {X 0,Y 495.784,Z 217.73,A -85,B 0,C 180,E1 -6236.976,E2 -6236.976} C_VEL
LIN {X 0,Y 495.767,Z 217.731,A -85,B 0,C 180,E1 -6239.746,E2 -6239.746} C_VEL
LIN {X 0,Y 495.769,Z 217.729,A -85,B 0,C 180,E1 -6242.594,E2 -6242.594} C_VEL
LIN {X 0,Y 495.746,Z 217.735,A -85,B 0,C 180,E1 -6245.538,E2 -6245.538} C_VEL
LIN {X 0,Y 495.763,Z 217.728,A -85,B 0,C 180,E1 -6248.768,E2 -6248.768} C_VEL
LIN {X 0,Y 495.757,Z 217.729,A -85,B 0,C 180,E1 -6251.781,E2 -6251.781} C_VEL
LIN {X 0,Y 495.75,Z 217.735,A -85,B 0,C 180,E1 -6255.139,E2 -6255.139} C_VEL
LIN {X 0,Y 495.756,Z 217.725,A -85,B 0,C 180,E1 -6258.219,E2 -6258.219} C_VEL
LIN {X 0,Y 495.75,Z 217.733,A -85,B 0,C 180,E1 -6261.408,E2 -6261.408} C_VEL
LIN {X 0,Y 495.755,Z 217.727,A -85,B 0,C 180,E1 -6264.463,E2 -6264.463} C_VEL
LIN {X 0,Y 495.767,Z 217.729,A -85,B 0,C 180,E1 -6267.406,E2 -6267.406} C_VEL
LIN {X 0,Y 495.766,Z 217.726,A -85,B 0,C 180,E1 -6270.254,E2 -6270.254} C_VEL
LIN {X 0,Y 495.823,Z 217.725,A -85,B 0,C 180,E1 -6273.251,E2 -6273.251} C_VEL
LIN {X 0,Y 495.747,Z 217.728,A -85,B 0,C 180,E1 -6275.725,E2 -6275.725} C_VEL
LIN {X 0,Y 495.741,Z 217.729,A -85,B 0,C 180,E1 -6278.371,E2 -6278.371} C_VEL
LIN {X 0,Y 495.783,Z 217.728,A -85,B 0,C 180,E1 -6280.972,E2 -6280.972} C_VEL
LIN {X 0,Y 495.777,Z 217.726,A -85,B 0,C 180,E1 -6283.53,E2 -6283.53} C_VEL
LIN {X 0,Y 495.796,Z 217.718,A -85,B 0,C 180,E1 -6286.056,E2 -6286.056} C_VEL
LIN {X 0,Y 495.851,Z 217.718,A -85,B 0,C 180,E1 -6288.555,E2 -6288.555} C_VEL
LIN {X 0,Y 495.872,Z 217.712,A -85,B 0,C 180,E1 -6291.852,E2 -6291.852} C_VEL
LIN {X 0,Y 495.888,Z 217.711,A -85,B 0,C 180,E1 -6294.306,E2 -6294.306} C_VEL
LIN {X 0,Y 495.993,Z 217.698,A -85,B 0,C 180,E1 -6297.564,E2 -6297.564} C_VEL
LIN {X 0,Y 496.004,Z 217.702,A -85,B 0,C 180,E1 -6300.812,E2 -6300.812} C_VEL
LIN {X 0,Y 495.839,Z 217.717,A -85,B 0,C 180,E1 -6303.25,E2 -6303.25} C_VEL
LIN {X 0,Y 495.859,Z 217.719,A -85,B 0,C 180,E1 -6306.511,E2 -6306.511} C_VEL
LIN {X 0,Y 495.841,Z 217.722,A -85,B 0,C 180,E1 -6308.97,E2 -6308.97} C_VEL
LIN {X 0,Y 495.827,Z 217.717,A -85,B 0,C 180,E1 -6312.035,E2 -6312.035} C_VEL
LIN {X 0,Y 495.823,Z 217.718,A -85,B 0,C 180,E1 -6315.452,E2 -6315.452} C_VEL
LIN {X 0,Y 495.806,Z 217.724,A -85,B 0,C 180,E1 -6318.248,E2 -6318.248} C_VEL
LIN {X 0,Y 495.774,Z 217.731,A -85,B 0,C 180,E1 -6320.757,E2 -6320.757} C_VEL
LIN {X 0,Y 495.746,Z 217.728,A -85,B 0,C 180,E1 -6323.388,E2 -6323.388} C_VEL
LIN {X 0,Y 495.759,Z 217.729,A -85,B 0,C 180,E1 -6326.07,E2 -6326.07} C_VEL
LIN {X 0,Y 495.743,Z 217.731,A -85,B 0,C 180,E1 -6328.817,E2 -6328.817} C_VEL
LIN {X 0,Y 495.755,Z 217.728,A -85,B 0,C 180,E1 -6331.725,E2 -6331.725} C_VEL
LIN {X 0,Y 495.761,Z 217.733,A -85,B 0,C 180,E1 -6334.693,E2 -6334.693} C_VEL
LIN {X 0,Y 495.707,Z 217.735,A -85,B 0,C 180,E1 -6337.564,E2 -6337.564} C_VEL
LIN {X 0,Y 495.743,Z 217.734,A -85,B 0,C 180,E1 -6340.045,E2 -6340.045} C_VEL
LIN {X 0,Y 495.704,Z 217.74,A -85,B 0,C 180,E1 -6342.886,E2 -6342.886} C_VEL
LIN {X 0,Y 495.801,Z 217.887,A -85,B 0,C 180,E1 -6344.241,E2 -6344.241} C_VEL
LIN {X 0,Y 496.673,Z 223.356,A -85,B 0,C 180,E1 -6345.301,E2 -6345.301} C_VEL
LIN {X 0,Y 496.342,Z 239.505,A -85,B 0,C 180,E1 -6348.279,E2 -6348.279} C_VEL
LIN {X 0,Y 496.274,Z 243.517,A -85,B 0,C 180,E1 -6349.021,E2 -6349.021} C_VEL
LIN {X 0,Y 498.635,Z 256.588,A -85,B 0,C 180,E1 -6349.294,E2 -6349.294} C_VEL
LIN {X 0,Y 498.143,Z 325.893,A -85,B 0,C 180,E1 -6350.303,E2 -6350.303} C_VEL
LIN {X 0,Y 497.476,Z 331.746,A -85,B 0,C 180,E1 -6350.364,E2 -6350.364} C_VEL
LIN {X 0,Y 491.796,Z 350.72,A -85,B 0,C 180,E1 -6350.489,E2 -6350.489} C_VEL
LIN {X 0,Y 491.027,Z 356.481,A -85,B 0,C 180,E1 -6350.608,E2 -6350.608} C_VEL
LIN {X 0,Y 490.756,Z 368.725,A -85,B 0,C 180,E1 -6351.008,E2 -6351.008} C_VEL
LIN {X 0,Y 490.459,Z 380.938,A -85,B 0,C 180,E1 -6351.572,E2 -6351.572} C_VEL
LIN {X 0,Y 490.122,Z 391.273,A -85,B 0,C 180,E1 -6352.193,E2 -6352.193} C_VEL
LIN {X 0,Y 489.732,Z 401.195,A -85,B 0,C 180,E1 -6352.934,E2 -6352.934} C_VEL
LIN {X 0,Y 489.298,Z 411.837,A -85,B 0,C 180,E1 -6353.921,E2 -6353.921} C_VEL
LIN {X 0,Y 488.928,Z 421.333,A -85,B 0,C 180,E1 -6355.019,E2 -6355.019} C_VEL
LIN {X 0,Y 488.575,Z 429.987,A -85,B 0,C 180,E1 -6356.253,E2 -6356.253} C_VEL
LIN {X 0,Y 488.36,Z 437.389,A -85,B 0,C 180,E1 -6357.584,E2 -6357.584} C_VEL
LIN {X 0,Y 488.165,Z 442.715,A -85,B 0,C 180,E1 -6358.783,E2 -6358.783} C_VEL
LIN {X 0,Y 488.032,Z 447.654,A -85,B 0,C 180,E1 -6360.222,E2 -6360.222} C_VEL
LIN {X 0,Y 487.912,Z 451.113,A -85,B 0,C 180,E1 -6361.619,E2 -6361.619} C_VEL
LIN {X 0,Y 487.826,Z 452.722,A -85,B 0,C 180,E1 -6362.547,E2 -6362.547} C_VEL
LIN {X 0,Y 487.81,Z 453.807,A -85,B 0,C 180,E1 -6363.473,E2 -6363.473} C_VEL
LIN {X 0,Y 487.778,Z 454.418,A -85,B 0,C 180,E1 -6364.39,E2 -6364.39} C_VEL
LIN {X 0,Y 487.809,Z 454.494,A -85,B 0,C 180,E1 -6365.304,E2 -6365.304} C_VEL
LIN {X 0,Y 487.755,Z 454.127,A -85,B 0,C 180,E1 -6366.206,E2 -6366.206} C_VEL
LIN {X 0,Y 487.803,Z 453.122,A -85,B 0,C 180,E1 -6367.232,E2 -6367.232} C_VEL
LIN {X 0,Y 487.931,Z 450.172,A -85,B 0,C 180,E1 -6368.894,E2 -6368.894} C_VEL
LIN {X 0,Y 488.097,Z 446.555,A -85,B 0,C 180,E1 -6370.222,E2 -6370.222} C_VEL
LIN {X 0,Y 488.197,Z 441.758,A -85,B 0,C 180,E1 -6371.536,E2 -6371.536} C_VEL
LIN {X 0,Y 488.354,Z 435.622,A -85,B 0,C 180,E1 -6372.841,E2 -6372.841} C_VEL
LIN {X 0,Y 488.684,Z 427.927,A -85,B 0,C 180,E1 -6374.142,E2 -6374.142} C_VEL
LIN {X 0,Y 488.996,Z 420.08,A -85,B 0,C 180,E1 -6375.22,E2 -6375.22} C_VEL
LIN {X 0,Y 489.332,Z 410.543,A -85,B 0,C 180,E1 -6376.292,E2 -6376.292} C_VEL
LIN {X 0,Y 489.758,Z 400.16,A -85,B 0,C 180,E1 -6377.229,E2 -6377.229} C_VEL
LIN {X 0,Y 490.161,Z 389.56,A -85,B 0,C 180,E1 -6378,E2 -6378} C_VEL
LIN {X 0,Y 490.526,Z 377.492,A -85,B 0,C 180,E1 -6378.691,E2 -6378.691} C_VEL
LIN {X 0,Y 490.81,Z 364.836,A -85,B 0,C 180,E1 -6379.22,E2 -6379.22} C_VEL
LIN {X 0,Y 491.063,Z 351.666,A -85,B 0,C 180,E1 -6379.59,E2 -6379.59} C_VEL
LIN {X 0,Y 491.803,Z 262.157,A -85,B 0,C 180,E1 -6380.933,E2 -6380.933} C_VEL
LIN {X 0,Y 491.511,Z 255.349,A -85,B 0,C 180,E1 -6381.045,E2 -6381.045} C_VEL
LIN {X 0,Y 489.31,Z 243.797,A -85,B 0,C 180,E1 -6381.297,E2 -6381.297} C_VEL
LIN {X 0,Y 489.72,Z 228.851,A -85,B 0,C 180,E1 -6384.234,E2 -6384.234} C_VEL
LIN {X 0,Y 489.72,Z 224.702,A -85,B 0,C 180,E1 -6385.06,E2 -6385.06} C_VEL
LIN {X 0,Y 488.697,Z 218.612,A -85,B 0,C 180,E1 -6386.341,E2 -6386.341} C_VEL
LIN {X 0,Y 488.946,Z 218.583,A -85,B 0,C 180,E1 -6387.528,E2 -6387.528} C_VEL
LIN {X 0,Y 488.944,Z 218.581,A -85,B 0,C 180,E1 -6390,E2 -6390} C_VEL
LIN {X 0,Y 488.946,Z 218.575,A -85,B 0,C 180,E1 -6392.471,E2 -6392.471} C_VEL
LIN {X 0,Y 488.819,Z 218.598,A -85,B 0,C 180,E1 -6395.776,E2 -6395.776} C_VEL
LIN {X 0,Y 488.782,Z 218.597,A -85,B 0,C 180,E1 -6398.267,E2 -6398.267} C_VEL
LIN {X 0,Y 488.808,Z 218.6,A -85,B 0,C 180,E1 -6401.612,E2 -6401.612} C_VEL
LIN {X 0,Y 488.758,Z 218.601,A -85,B 0,C 180,E1 -6405,E2 -6405} C_VEL
LIN {X 0,Y 488.746,Z 218.601,A -85,B 0,C 180,E1 -6408.442,E2 -6408.442} C_VEL
LIN {X 0,Y 488.709,Z 218.608,A -85,B 0,C 180,E1 -6411.07,E2 -6411.07} C_VEL
LIN {X 0,Y 488.673,Z 218.616,A -85,B 0,C 180,E1 -6413.746,E2 -6413.746} C_VEL
LIN {X 0,Y 488.726,Z 218.606,A -85,B 0,C 180,E1 -6416.928,E2 -6416.928} C_VEL
LIN {X 0,Y 488.724,Z 218.605,A -85,B 0,C 180,E1 -6420.219,E2 -6420.219} C_VEL
LIN {X 0,Y 488.735,Z 218.608,A -85,B 0,C 180,E1 -6423.484,E2 -6423.484} C_VEL
LIN {X 0,Y 488.673,Z 218.611,A -85,B 0,C 180,E1 -6426.353,E2 -6426.353} C_VEL
LIN {X 0,Y 488.7,Z 218.611,A -85,B 0,C 180,E1 -6429.254,E2 -6429.254} C_VEL
LIN {X 0,Y 488.688,Z 218.61,A -85,B 0,C 180,E1 -6432.525,E2 -6432.525} C_VEL
LIN {X 0,Y 488.701,Z 218.611,A -85,B 0,C 180,E1 -6435.197,E2 -6435.197} C_VEL
LIN {X 0,Y 488.706,Z 218.608,A -85,B 0,C 180,E1 -6438.584,E2 -6438.584} C_VEL
LIN {X 0,Y 488.703,Z 218.61,A -85,B 0,C 180,E1 -6440.947,E2 -6440.947} C_VEL
LIN {X 0,Y 488.682,Z 218.612,A -85,B 0,C 180,E1 -6443.868,E2 -6443.868} C_VEL
LIN {X 0,Y 488.737,Z 218.607,A -85,B 0,C 180,E1 -6446.877,E2 -6446.877} C_VEL
LIN {X 0,Y 488.722,Z 218.607,A -85,B 0,C 180,E1 -6449.78,E2 -6449.78} C_VEL
LIN {X 0,Y 488.79,Z 218.6,A -85,B 0,C 180,E1 -6453.056,E2 -6453.056} C_VEL
LIN {X 0,Y 488.692,Z 218.609,A -85,B 0,C 180,E1 -6456.254,E2 -6456.254} C_VEL
LIN {X 0,Y 488.744,Z 218.606,A -85,B 0,C 180,E1 -6459.175,E2 -6459.175} C_VEL
LIN {X 0,Y 488.757,Z 218.604,A -85,B 0,C 180,E1 -6461.627,E2 -6461.627} C_VEL
LIN {X 0,Y 488.759,Z 218.604,A -85,B 0,C 180,E1 -6464.999,E2 -6464.999} C_VEL
LIN {X 0,Y 488.803,Z 218.596,A -85,B 0,C 180,E1 -6468.387,E2 -6468.387} C_VEL
LIN {X 0,Y 488.815,Z 218.595,A -85,B 0,C 180,E1 -6471.733,E2 -6471.733} C_VEL
LIN {X 0,Y 488.855,Z 218.589,A -85,B 0,C 180,E1 -6474.224,E2 -6474.224} C_VEL
LIN {X 0,Y 488.959,Z 218.578,A -85,B 0,C 180,E1 -6477.529,E2 -6477.529} C_VEL
LIN {X 0,Y 488.967,Z 218.575,A -85,B 0,C 180,E1 -6480,E2 -6480} C_VEL
LIN {X 0,Y 488.959,Z 218.578,A -85,B 0,C 180,E1 -6482.471,E2 -6482.471} C_VEL
LIN {X 0,Y 488.855,Z 218.589,A -85,B 0,C 180,E1 -6485.776,E2 -6485.776} C_VEL
LIN {X 0,Y 488.814,Z 218.595,A -85,B 0,C 180,E1 -6488.266,E2 -6488.266} C_VEL
LIN {X 0,Y 488.803,Z 218.596,A -85,B 0,C 180,E1 -6491.612,E2 -6491.612} C_VEL
LIN {X 0,Y 488.759,Z 218.604,A -85,B 0,C 180,E1 -6495,E2 -6495} C_VEL
LIN {X 0,Y 488.752,Z 218.604,A -85,B 0,C 180,E1 -6498.442,E2 -6498.442} C_VEL
LIN {X 0,Y 488.705,Z 218.61,A -85,B 0,C 180,E1 -6501.071,E2 -6501.071} C_VEL
LIN {X 0,Y 488.691,Z 218.609,A -85,B 0,C 180,E1 -6503.746,E2 -6503.746} C_VEL
LIN {X 0,Y 488.789,Z 218.6,A -85,B 0,C 180,E1 -6506.944,E2 -6506.944} C_VEL
LIN {X 0,Y 488.707,Z 218.61,A -85,B 0,C 180,E1 -6510.363,E2 -6510.363} C_VEL
LIN {X 0,Y 488.733,Z 218.604,A -85,B 0,C 180,E1 -6513.485,E2 -6513.485} C_VEL
LIN {X 0,Y 488.686,Z 218.612,A -85,B 0,C 180,E1 -6516.356,E2 -6516.356} C_VEL
LIN {X 0,Y 488.699,Z 218.609,A -85,B 0,C 180,E1 -6519.255,E2 -6519.255} C_VEL
LIN {X 0,Y 488.705,Z 218.606,A -85,B 0,C 180,E1 -6521.6,E2 -6521.6} C_VEL
LIN {X 0,Y 488.711,Z 218.61,A -85,B 0,C 180,E1 -6524.802,E2 -6524.802} C_VEL
LIN {X 0,Y 488.691,Z 218.608,A -85,B 0,C 180,E1 -6527.475,E2 -6527.475} C_VEL
LIN {X 0,Y 488.732,Z 218.602,A -85,B 0,C 180,E1 -6529.677,E2 -6529.677} C_VEL
LIN {X 0,Y 488.67,Z 218.614,A -85,B 0,C 180,E1 -6532.841,E2 -6532.841} C_VEL
LIN {X 0,Y 488.73,Z 218.603,A -85,B 0,C 180,E1 -6535.888,E2 -6535.888} C_VEL
LIN {X 0,Y 488.693,Z 218.614,A -85,B 0,C 180,E1 -6538.821,E2 -6538.821} C_VEL
LIN {X 0,Y 488.742,Z 218.603,A -85,B 0,C 180,E1 -6541.671,E2 -6541.671} C_VEL
LIN {X 0,Y 488.708,Z 218.615,A -85,B 0,C 180,E1 -6544.442,E2 -6544.442} C_VEL
LIN {X 0,Y 488.702,Z 218.668,A -85,B 0,C 180,E1 -6544.959,E2 -6544.959} C_VEL
LIN {X 0,Y 490.605,Z 228.916,A -85,B 0,C 180,E1 -6546.865,E2 -6546.865} C_VEL
LIN {X 0,Y 490.099,Z 243.764,A -85,B 0,C 180,E1 -6549.432,E2 -6549.432} C_VEL
LIN {X 0,Y 489.5,Z 261.5,A -85,B 0,C 180,E1 -6552.452,E2 -6552.452} C_VEL
LIN {X 0,Y 489.252,Z 269.096,A -85,B 0,C 180,E1 -6553.733,E2 -6553.733} C_VEL
LIN {X 0,Y 491.665,Z 284.849,A -85,B 0,C 180,E1 -6554.052,E2 -6554.052} C_VEL
LIN {X 0,Y 491.034,Z 377.637,A -85,B 0,C 180,E1 -6555.442,E2 -6555.442} C_VEL
LIN {X 0,Y 490.711,Z 391.521,A -85,B 0,C 180,E1 -6555.829,E2 -6555.829} C_VEL
LIN {X 0,Y 490.361,Z 404.474,A -85,B 0,C 180,E1 -6556.374,E2 -6556.374} C_VEL
LIN {X 0,Y 489.977,Z 416.262,A -85,B 0,C 180,E1 -6557.05,E2 -6557.05} C_VEL
LIN {X 0,Y 489.599,Z 427.619,A -85,B 0,C 180,E1 -6557.882,E2 -6557.882} C_VEL
LIN {X 0,Y 489.203,Z 437.864,A -85,B 0,C 180,E1 -6558.817,E2 -6558.817} C_VEL
LIN {X 0,Y 488.789,Z 447.068,A -85,B 0,C 180,E1 -6559.855,E2 -6559.855} C_VEL
LIN {X 0,Y 488.448,Z 456.032,A -85,B 0,C 180,E1 -6561.102,E2 -6561.102} C_VEL
LIN {X 0,Y 488.21,Z 463.248,A -85,B 0,C 180,E1 -6562.348,E2 -6562.348} C_VEL
LIN {X 0,Y 488.093,Z 468.521,A -85,B 0,C 180,E1 -6563.477,E2 -6563.477} C_VEL
LIN {X 0,Y 488.017,Z 472.85,A -85,B 0,C 180,E1 -6564.629,E2 -6564.629} C_VEL
LIN {X 0,Y 487.927,Z 476.463,A -85,B 0,C 180,E1 -6565.87,E2 -6565.87} C_VEL
LIN {X 0,Y 487.964,Z 478.329,A -85,B 0,C 180,E1 -6566.697,E2 -6566.697} C_VEL
LIN {X 0,Y 487.891,Z 480.721,A -85,B 0,C 180,E1 -6568.349,E2 -6568.349} C_VEL
LIN {X 0,Y 487.821,Z 481.54,A -85,B 0,C 180,E1 -6570,E2 -6570} C_VEL
LIN {X 0,Y 487.891,Z 480.712,A -85,B 0,C 180,E1 -6571.651,E2 -6571.651} C_VEL
LIN {X 0,Y 487.909,Z 479.712,A -85,B 0,C 180,E1 -6572.477,E2 -6572.477} C_VEL
LIN {X 0,Y 487.964,Z 478.311,A -85,B 0,C 180,E1 -6573.303,E2 -6573.303} C_VEL
LIN {X 0,Y 487.919,Z 475.363,A -85,B 0,C 180,E1 -6574.544,E2 -6574.544} C_VEL
LIN {X 0,Y 488.02,Z 471.377,A -85,B 0,C 180,E1 -6575.786,E2 -6575.786} C_VEL
LIN {X 0,Y 488.18,Z 465.245,A -85,B 0,C 180,E1 -6577.237,E2 -6577.237} C_VEL
LIN {X 0,Y 488.36,Z 458.546,A -85,B 0,C 180,E1 -6578.483,E2 -6578.483} C_VEL
LIN {X 0,Y 488.665,Z 450.235,A -85,B 0,C 180,E1 -6579.729,E2 -6579.729} C_VEL
LIN {X 0,Y 488.993,Z 441.711,A -85,B 0,C 180,E1 -6580.769,E2 -6580.769} C_VEL
LIN {X 0,Y 489.432,Z 431.18,A -85,B 0,C 180,E1 -6581.807,E2 -6581.807} C_VEL
LIN {X 0,Y 489.818,Z 419.454,A -85,B 0,C 180,E1 -6582.735,E2 -6582.735} C_VEL
LIN {X 0,Y 490.248,Z 407.381,A -85,B 0,C 180,E1 -6583.471,E2 -6583.471} C_VEL
LIN {X 0,Y 490.63,Z 394.953,A -85,B 0,C 180,E1 -6584.041,E2 -6584.041} C_VEL
LIN {X 0,Y 490.974,Z 382.13,A -85,B 0,C 180,E1 -6584.454,E2 -6584.454} C_VEL
LIN {X 0,Y 491.213,Z 366.765,A -85,B 0,C 180,E1 -6584.738,E2 -6584.738} C_VEL
LIN {X 0,Y 491.601,Z 283.84,A -85,B 0,C 180,E1 -6585.967,E2 -6585.967} C_VEL
LIN {X 0,Y 489.239,Z 268.832,A -85,B 0,C 180,E1 -6586.277,E2 -6586.277} C_VEL
LIN {X 0,Y 489.785,Z 250.981,A -85,B 0,C 180,E1 -6589.271,E2 -6589.271} C_VEL
LIN {X 0,Y 490.389,Z 232.999,A -85,B 0,C 180,E1 -6592.32,E2 -6592.32} C_VEL
LIN {X 0,Y 490.485,Z 228.508,A -85,B 0,C 180,E1 -6593.092,E2 -6593.092} C_VEL
LIN {X 0,Y 488.687,Z 218.614,A -85,B 0,C 180,E1 -6594.925,E2 -6594.925} C_VEL
LIN {X 0,Y 488.731,Z 218.609,A -85,B 0,C 180,E1 -6597.398,E2 -6597.398} C_VEL
LIN {X 0,Y 488.71,Z 218.606,A -85,B 0,C 180,E1 -6600.362,E2 -6600.362} C_VEL
LIN {X 0,Y 488.736,Z 218.61,A -85,B 0,C 180,E1 -6603.484,E2 -6603.484} C_VEL
LIN {X 0,Y 488.674,Z 218.61,A -85,B 0,C 180,E1 -6606.353,E2 -6606.353} C_VEL
LIN {X 0,Y 488.701,Z 218.614,A -85,B 0,C 180,E1 -6609.254,E2 -6609.254} C_VEL
LIN {X 0,Y 488.707,Z 218.609,A -85,B 0,C 180,E1 -6611.6,E2 -6611.6} C_VEL
LIN {X 0,Y 488.712,Z 218.608,A -85,B 0,C 180,E1 -6614.801,E2 -6614.801} C_VEL
LIN {X 0,Y 488.692,Z 218.611,A -85,B 0,C 180,E1 -6617.474,E2 -6617.474} C_VEL
LIN {X 0,Y 488.733,Z 218.605,A -85,B 0,C 180,E1 -6619.676,E2 -6619.676} C_VEL
LIN {X 0,Y 488.682,Z 218.612,A -85,B 0,C 180,E1 -6622.841,E2 -6622.841} C_VEL
LIN {X 0,Y 488.734,Z 218.602,A -85,B 0,C 180,E1 -6625.887,E2 -6625.887} C_VEL
LIN {X 0,Y 488.691,Z 218.609,A -85,B 0,C 180,E1 -6628.82,E2 -6628.82} C_VEL
LIN {X 0,Y 488.744,Z 218.6,A -85,B 0,C 180,E1 -6631.671,E2 -6631.671} C_VEL
LIN {X 0,Y 488.746,Z 218.601,A -85,B 0,C 180,E1 -6634.444,E2 -6634.444} C_VEL
LIN {X 0,Y 488.722,Z 218.608,A -85,B 0,C 180,E1 -6637.153,E2 -6637.153} C_VEL
LIN {X 0,Y 488.724,Z 218.603,A -85,B 0,C 180,E1 -6639.81,E2 -6639.81} C_VEL
LIN {X 0,Y 488.728,Z 218.602,A -85,B 0,C 180,E1 -6642.423,E2 -6642.423} C_VEL
LIN {X 0,Y 488.761,Z 218.602,A -85,B 0,C 180,E1 -6645,E2 -6645} C_VEL
LIN {X 0,Y 488.805,Z 218.594,A -85,B 0,C 180,E1 -6648.388,E2 -6648.388} C_VEL
LIN {X 0,Y 488.816,Z 218.591,A -85,B 0,C 180,E1 -6651.734,E2 -6651.734} C_VEL
LIN {X 0,Y 488.847,Z 218.588,A -85,B 0,C 180,E1 -6654.224,E2 -6654.224} C_VEL
LIN {X 0,Y 488.961,Z 218.575,A -85,B 0,C 180,E1 -6657.529,E2 -6657.529} C_VEL
LIN {X 0,Y 488.953,Z 218.58,A -85,B 0,C 180,E1 -6660.824,E2 -6660.824} C_VEL
LIN {X 0,Y 488.96,Z 218.578,A -85,B 0,C 180,E1 -6662.471,E2 -6662.471} C_VEL
LIN {X 0,Y 488.846,Z 218.588,A -85,B 0,C 180,E1 -6665.776,E2 -6665.776} C_VEL
LIN {X 0,Y 488.817,Z 218.592,A -85,B 0,C 180,E1 -6668.266,E2 -6668.266} C_VEL
LIN {X 0,Y 488.805,Z 218.591,A -85,B 0,C 180,E1 -6671.613,E2 -6671.613} C_VEL
LIN {X 0,Y 488.764,Z 218.601,A -85,B 0,C 180,E1 -6675,E2 -6675} C_VEL
LIN {X 0,Y 488.755,Z 218.605,A -85,B 0,C 180,E1 -6678.442,E2 -6678.442} C_VEL
LIN {X 0,Y 488.706,Z 218.608,A -85,B 0,C 180,E1 -6681.071,E2 -6681.071} C_VEL
LIN {X 0,Y 488.683,Z 218.608,A -85,B 0,C 180,E1 -6683.746,E2 -6683.746} C_VEL
LIN {X 0,Y 488.724,Z 218.608,A -85,B 0,C 180,E1 -6686.928,E2 -6686.928} C_VEL
LIN {X 0,Y 488.723,Z 218.606,A -85,B 0,C 180,E1 -6690.22,E2 -6690.22} C_VEL
LIN {X 0,Y 488.729,Z 218.605,A -85,B 0,C 180,E1 -6693.483,E2 -6693.483} C_VEL
LIN {X 0,Y 488.668,Z 218.62,A -85,B 0,C 180,E1 -6696.352,E2 -6696.352} C_VEL
LIN {X 0,Y 488.687,Z 218.61,A -85,B 0,C 180,E1 -6699.256,E2 -6699.256} C_VEL
LIN {X 0,Y 488.667,Z 218.618,A -85,B 0,C 180,E1 -6702.529,E2 -6702.529} C_VEL
LIN {X 0,Y 488.75,Z 218.753,A -85,B 0,C 180,E1 -6704.085,E2 -6704.085} C_VEL
LIN {X 0,Y 489.689,Z 225.077,A -85,B 0,C 180,E1 -6705.312,E2 -6705.312} C_VEL
LIN {X 0,Y 489.352,Z 241.195,A -85,B 0,C 180,E1 -6708.316,E2 -6708.316} C_VEL
LIN {X 0,Y 489.312,Z 243.622,A -85,B 0,C 180,E1 -6708.77,E2 -6708.77} C_VEL
LIN {X 0,Y 491.76,Z 256.861,A -85,B 0,C 180,E1 -6709.068,E2 -6709.068} C_VEL
LIN {X 0,Y 491.078,Z 351.737,A -85,B 0,C 180,E1 -6710.495,E2 -6710.495} C_VEL
LIN {X 0,Y 491.027,Z 356.481,A -85,B 0,C 180,E1 -6710.608,E2 -6710.608} C_VEL
LIN {X 0,Y 490.237,Z 360.34,A -85,B 0,C 180,E1 -6710.694,E2 -6710.694} C_VEL
LIN {X 0,Y 484.383,Z 372.336,A -85,B 0,C 180,E1 -6710.961,E2 -6710.961} C_VEL
LIN {X 0,Y 483.726,Z 376.018,A -85,B 0,C 180,E1 -6711.115,E2 -6711.115} C_VEL
LIN {X 0,Y 483.341,Z 387.409,A -85,B 0,C 180,E1 -6711.738,E2 -6711.738} C_VEL
LIN {X 0,Y 482.886,Z 399.153,A -85,B 0,C 180,E1 -6712.574,E2 -6712.574} C_VEL
LIN {X 0,Y 482.424,Z 410.334,A -85,B 0,C 180,E1 -6713.584,E2 -6713.584} C_VEL
LIN {X 0,Y 482.054,Z 419.236,A -85,B 0,C 180,E1 -6714.577,E2 -6714.577} C_VEL
LIN {X 0,Y 481.648,Z 428.258,A -85,B 0,C 180,E1 -6715.822,E2 -6715.822} C_VEL
LIN {X 0,Y 481.368,Z 435.46,A -85,B 0,C 180,E1 -6717.054,E2 -6717.054} C_VEL
LIN {X 0,Y 481.157,Z 441.228,A -85,B 0,C 180,E1 -6718.276,E2 -6718.276} C_VEL
LIN {X 0,Y 481.037,Z 445.973,A -85,B 0,C 180,E1 -6719.542,E2 -6719.542} C_VEL
LIN {X 0,Y 480.854,Z 450.455,A -85,B 0,C 180,E1 -6721.163,E2 -6721.163} C_VEL
LIN {X 0,Y 480.758,Z 452.291,A -85,B 0,C 180,E1 -6722.109,E2 -6722.109} C_VEL
LIN {X 0,Y 480.73,Z 453.673,A -85,B 0,C 180,E1 -6723.099,E2 -6723.099} C_VEL
LIN {X 0,Y 480.682,Z 454.4,A -85,B 0,C 180,E1 -6723.984,E2 -6723.984} C_VEL
LIN {X 0,Y 480.681,Z 454.736,A -85,B 0,C 180,E1 -6725.026,E2 -6725.026} C_VEL
LIN {X 0,Y 480.668,Z 454.547,A -85,B 0,C 180,E1 -6725.833,E2 -6725.833} C_VEL
LIN {X 0,Y 480.71,Z 453.556,A -85,B 0,C 180,E1 -6727.083,E2 -6727.083} C_VEL
LIN {X 0,Y 480.815,Z 451.181,A -85,B 0,C 180,E1 -6728.567,E2 -6728.567} C_VEL
LIN {X 0,Y 480.962,Z 447.872,A -85,B 0,C 180,E1 -6729.916,E2 -6729.916} C_VEL
LIN {X 0,Y 481.097,Z 443.41,A -85,B 0,C 180,E1 -6731.253,E2 -6731.253} C_VEL
LIN {X 0,Y 481.26,Z 437.685,A -85,B 0,C 180,E1 -6732.58,E2 -6732.58} C_VEL
LIN {X 0,Y 481.546,Z 430.499,A -85,B 0,C 180,E1 -6733.901,E2 -6733.901} C_VEL
LIN {X 0,Y 481.857,Z 423.126,A -85,B 0,C 180,E1 -6734.996,E2 -6734.996} C_VEL
LIN {X 0,Y 482.277,Z 413.161,A -85,B 0,C 180,E1 -6736.195,E2 -6736.195} C_VEL
LIN {X 0,Y 482.703,Z 402.877,A -85,B 0,C 180,E1 -6737.193,E2 -6737.193} C_VEL
LIN {X 0,Y 483.175,Z 391.963,A -85,B 0,C 180,E1 -6738.037,E2 -6738.037} C_VEL
LIN {X 0,Y 483.588,Z 379.449,A -85,B 0,C 180,E1 -6738.791,E2 -6738.791} C_VEL
LIN {X 0,Y 483.9,Z 367.584,A -85,B 0,C 180,E1 -6739.329,E2 -6739.329} C_VEL
LIN {X 0,Y 484.172,Z 354.693,A -85,B 0,C 180,E1 -6739.731,E2 -6739.731} C_VEL
LIN {X 0,Y 484.349,Z 336.535,A -85,B 0,C 180,E1 -6740.052,E2 -6740.052} C_VEL
LIN {X 0,Y 484.916,Z 257.608,A -85,B 0,C 180,E1 -6741.234,E2 -6741.234} C_VEL
LIN {X 0,Y 482.306,Z 243.901,A -85,B 0,C 180,E1 -6741.55,E2 -6741.55} C_VEL
LIN {X 0,Y 482.732,Z 230.808,A -85,B 0,C 180,E1 -6744.151,E2 -6744.151} C_VEL
LIN {X 0,Y 482.72,Z 225.63,A -85,B 0,C 180,E1 -6745.198,E2 -6745.198} C_VEL
LIN {X 0,Y 481.706,Z 219.483,A -85,B 0,C 180,E1 -6746.497,E2 -6746.497} C_VEL
LIN {X 0,Y 481.911,Z 219.46,A -85,B 0,C 180,E1 -6747.492,E2 -6747.492} C_VEL
LIN {X 0,Y 481.914,Z 219.456,A -85,B 0,C 180,E1 -6750,E2 -6750} C_VEL
LIN {X 0,Y 481.912,Z 219.452,A -85,B 0,C 180,E1 -6752.507,E2 -6752.507} C_VEL
LIN {X 0,Y 481.78,Z 219.473,A -85,B 0,C 180,E1 -6755.861,E2 -6755.861} C_VEL
LIN {X 0,Y 481.738,Z 219.474,A -85,B 0,C 180,E1 -6758.389,E2 -6758.389} C_VEL
LIN {X 0,Y 481.754,Z 219.478,A -85,B 0,C 180,E1 -6761.785,E2 -6761.785} C_VEL
LIN {X 0,Y 481.741,Z 219.476,A -85,B 0,C 180,E1 -6765.224,E2 -6765.224} C_VEL
LIN {X 0,Y 481.708,Z 219.478,A -85,B 0,C 180,E1 -6768.722,E2 -6768.722} C_VEL
LIN {X 0,Y 481.647,Z 219.49,A -85,B 0,C 180,E1 -6771.394,E2 -6771.394} C_VEL
LIN {X 0,Y 481.651,Z 219.487,A -85,B 0,C 180,E1 -6774.114,E2 -6774.114} C_VEL
LIN {X 0,Y 481.696,Z 219.482,A -85,B 0,C 180,E1 -6777.126,E2 -6777.126} C_VEL
LIN {X 0,Y 481.674,Z 219.487,A -85,B 0,C 180,E1 -6779.741,E2 -6779.741} C_VEL
LIN {X 0,Y 481.673,Z 219.484,A -85,B 0,C 180,E1 -6782.674,E2 -6782.674} C_VEL
LIN {X 0,Y 481.661,Z 219.487,A -85,B 0,C 180,E1 -6785.203,E2 -6785.203} C_VEL
LIN {X 0,Y 481.67,Z 219.486,A -85,B 0,C 180,E1 -6788.859,E2 -6788.859} C_VEL
LIN {X 0,Y 481.646,Z 219.488,A -85,B 0,C 180,E1 -6791.912,E2 -6791.912} C_VEL
LIN {X 0,Y 481.653,Z 219.486,A -85,B 0,C 180,E1 -6794.458,E2 -6794.458} C_VEL
LIN {X 0,Y 481.646,Z 219.489,A -85,B 0,C 180,E1 -6797.839,E2 -6797.839} C_VEL
LIN {X 0,Y 481.66,Z 219.486,A -85,B 0,C 180,E1 -6800.654,E2 -6800.654} C_VEL
LIN {X 0,Y 481.629,Z 219.493,A -85,B 0,C 180,E1 -6803.375,E2 -6803.375} C_VEL
LIN {X 0,Y 481.708,Z 219.479,A -85,B 0,C 180,E1 -6806.33,E2 -6806.33} C_VEL
LIN {X 0,Y 481.649,Z 219.491,A -85,B 0,C 180,E1 -6809.417,E2 -6809.417} C_VEL
LIN {X 0,Y 481.698,Z 219.481,A -85,B 0,C 180,E1 -6812.168,E2 -6812.168} C_VEL
LIN {X 0,Y 481.716,Z 219.481,A -85,B 0,C 180,E1 -6814.97,E2 -6814.97} C_VEL
LIN {X 0,Y 481.648,Z 219.489,A -85,B 0,C 180,E1 -6817.705,E2 -6817.705} C_VEL
LIN {X 0,Y 481.703,Z 219.481,A -85,B 0,C 180,E1 -6820.393,E2 -6820.393} C_VEL
LIN {X 0,Y 481.686,Z 219.485,A -85,B 0,C 180,E1 -6823.034,E2 -6823.034} C_VEL
LIN {X 0,Y 481.687,Z 219.484,A -85,B 0,C 180,E1 -6825.639,E2 -6825.639} C_VEL
LIN {X 0,Y 481.748,Z 219.475,A -85,B 0,C 180,E1 -6828.215,E2 -6828.215} C_VEL
LIN {X 0,Y 481.76,Z 219.475,A -85,B 0,C 180,E1 -6831.612,E2 -6831.612} C_VEL
LIN {X 0,Y 481.816,Z 219.466,A -85,B 0,C 180,E1 -6834.139,E2 -6834.139} C_VEL
LIN {X 0,Y 481.926,Z 219.455,A -85,B 0,C 180,E1 -6837.492,E2 -6837.492} C_VEL
LIN {X 0,Y 481.938,Z 219.451,A -85,B 0,C 180,E1 -6840,E2 -6840} C_VEL
LIN {X 0,Y 481.926,Z 219.455,A -85,B 0,C 180,E1 -6842.507,E2 -6842.507} C_VEL
LIN {X 0,Y 481.816,Z 219.466,A -85,B 0,C 180,E1 -6845.86,E2 -6845.86} C_VEL
LIN {X 0,Y 481.76,Z 219.475,A -85,B 0,C 180,E1 -6848.388,E2 -6848.388} C_VEL
LIN {X 0,Y 481.748,Z 219.474,A -85,B 0,C 180,E1 -6851.785,E2 -6851.785} C_VEL
LIN {X 0,Y 481.74,Z 219.477,A -85,B 0,C 180,E1 -6855.224,E2 -6855.224} C_VEL
LIN {X 0,Y 481.71,Z 219.484,A -85,B 0,C 180,E1 -6858.722,E2 -6858.722} C_VEL
LIN {X 0,Y 481.645,Z 219.489,A -85,B 0,C 180,E1 -6861.395,E2 -6861.395} C_VEL
LIN {X 0,Y 481.675,Z 219.484,A -85,B 0,C 180,E1 -6864.113,E2 -6864.113} C_VEL
LIN {X 0,Y 481.744,Z 219.476,A -85,B 0,C 180,E1 -6867.139,E2 -6867.139} C_VEL
LIN {X 0,Y 481.676,Z 219.483,A -85,B 0,C 180,E1 -6869.741,E2 -6869.741} C_VEL
LIN {X 0,Y 481.67,Z 219.489,A -85,B 0,C 180,E1 -6872.674,E2 -6872.674} C_VEL
LIN {X 0,Y 481.64,Z 219.487,A -85,B 0,C 180,E1 -6875.709,E2 -6875.709} C_VEL
LIN {X 0,Y 481.669,Z 219.487,A -85,B 0,C 180,E1 -6878.859,E2 -6878.859} C_VEL
LIN {X 0,Y 481.651,Z 219.486,A -85,B 0,C 180,E1 -6881.913,E2 -6881.913} C_VEL
LIN {X 0,Y 481.658,Z 219.489,A -85,B 0,C 180,E1 -6884.458,E2 -6884.458} C_VEL
LIN {X 0,Y 481.647,Z 219.486,A -85,B 0,C 180,E1 -6887.84,E2 -6887.84} C_VEL
LIN {X 0,Y 481.679,Z 219.488,A -85,B 0,C 180,E1 -6890.652,E2 -6890.652} C_VEL
LIN {X 0,Y 481.621,Z 219.489,A -85,B 0,C 180,E1 -6893.378,E2 -6893.378} C_VEL
LIN {X 0,Y 481.71,Z 219.482,A -85,B 0,C 180,E1 -6896.33,E2 -6896.33} C_VEL
LIN {X 0,Y 481.651,Z 219.486,A -85,B 0,C 180,E1 -6899.418,E2 -6899.418} C_VEL
LIN {X 0,Y 481.692,Z 219.485,A -85,B 0,C 180,E1 -6902.168,E2 -6902.168} C_VEL
LIN {X 0,Y 481.666,Z 219.611,A -85,B 0,C 180,E1 -6904.776,E2 -6904.776} C_VEL
LIN {X 0,Y 483.569,Z 229.411,A -85,B 0,C 180,E1 -6906.633,E2 -6906.633} C_VEL
LIN {X 0,Y 483.412,Z 238.399,A -85,B 0,C 180,E1 -6908.222,E2 -6908.222} C_VEL
LIN {X 0,Y 482.681,Z 257.499,A -85,B 0,C 180,E1 -6911.538,E2 -6911.538} C_VEL
LIN {X 0,Y 482.262,Z 268.979,A -85,B 0,C 180,E1 -6913.497,E2 -6913.497} C_VEL
LIN {X 0,Y 484.847,Z 286.355,A -85,B 0,C 180,E1 -6913.85,E2 -6913.85} C_VEL
LIN {X 0,Y 484.183,Z 377.287,A -85,B 0,C 180,E1 -6915.231,E2 -6915.231} C_VEL
LIN {X 0,Y 483.867,Z 390.46,A -85,B 0,C 180,E1 -6915.598,E2 -6915.598} C_VEL
LIN {X 0,Y 483.497,Z 403.146,A -85,B 0,C 180,E1 -6916.123,E2 -6916.123} C_VEL
LIN {X 0,Y 483.106,Z 414.43,A -85,B 0,C 180,E1 -6916.755,E2 -6916.755} C_VEL
LIN {X 0,Y 482.648,Z 426.143,A -85,B 0,C 180,E1 -6917.602,E2 -6917.602} C_VEL
LIN {X 0,Y 482.218,Z 436.583,A -85,B 0,C 180,E1 -6918.547,E2 -6918.547} C_VEL
LIN {X 0,Y 481.82,Z 445.16,A -85,B 0,C 180,E1 -6919.495,E2 -6919.495} C_VEL
LIN {X 0,Y 481.484,Z 453.073,A -85,B 0,C 180,E1 -6920.549,E2 -6920.549} C_VEL
LIN {X 0,Y 481.226,Z 460.801,A -85,B 0,C 180,E1 -6921.814,E2 -6921.814} C_VEL
LIN {X 0,Y 481.012,Z 467.915,A -85,B 0,C 180,E1 -6923.288,E2 -6923.288} C_VEL
LIN {X 0,Y 480.93,Z 472.649,A -85,B 0,C 180,E1 -6924.55,E2 -6924.55} C_VEL
LIN {X 0,Y 480.827,Z 476.264,A -85,B 0,C 180,E1 -6925.809,E2 -6925.809} C_VEL
LIN {X 0,Y 480.888,Z 478.132,A -85,B 0,C 180,E1 -6926.649,E2 -6926.649} C_VEL
LIN {X 0,Y 480.823,Z 479.529,A -85,B 0,C 180,E1 -6927.487,E2 -6927.487} C_VEL
LIN {X 0,Y 480.76,Z 481.13,A -85,B 0,C 180,E1 -6929.163,E2 -6929.163} C_VEL
LIN {X 0,Y 480.745,Z 481.345,A -85,B 0,C 180,E1 -6930,E2 -6930} C_VEL
LIN {X 0,Y 480.76,Z 481.126,A -85,B 0,C 180,E1 -6930.838,E2 -6930.838} C_VEL
LIN {X 0,Y 480.823,Z 479.515,A -85,B 0,C 180,E1 -6932.513,E2 -6932.513} C_VEL
LIN {X 0,Y 480.888,Z 478.113,A -85,B 0,C 180,E1 -6933.351,E2 -6933.351} C_VEL
LIN {X 0,Y 480.838,Z 475.164,A -85,B 0,C 180,E1 -6934.611,E2 -6934.611} C_VEL
LIN {X 0,Y 480.925,Z 471.175,A -85,B 0,C 180,E1 -6935.871,E2 -6935.871} C_VEL
LIN {X 0,Y 481.105,Z 465.042,A -85,B 0,C 180,E1 -6937.344,E2 -6937.344} C_VEL
LIN {X 0,Y 481.318,Z 458.342,A -85,B 0,C 180,E1 -6938.608,E2 -6938.608} C_VEL
LIN {X 0,Y 481.635,Z 450.031,A -85,B 0,C 180,E1 -6939.873,E2 -6939.873} C_VEL
LIN {X 0,Y 482.011,Z 441.508,A -85,B 0,C 180,E1 -6940.926,E2 -6940.926} C_VEL
LIN {X 0,Y 482.45,Z 430.997,A -85,B 0,C 180,E1 -6941.979,E2 -6941.979} C_VEL
LIN {X 0,Y 482.865,Z 419.628,A -85,B 0,C 180,E1 -6942.894,E2 -6942.894} C_VEL
LIN {X 0,Y 483.258,Z 409.13,A -85,B 0,C 180,E1 -6943.562,E2 -6943.562} C_VEL
LIN {X 0,Y 483.656,Z 397.354,A -85,B 0,C 180,E1 -6944.141,E2 -6944.141} C_VEL
LIN {X 0,Y 484.048,Z 383.787,A -85,B 0,C 180,E1 -6944.612,E2 -6944.612} C_VEL
LIN {X 0,Y 484.319,Z 370.128,A -85,B 0,C 180,E1 -6944.899,E2 -6944.899} C_VEL
LIN {X 0,Y 484.694,Z 284.006,A -85,B 0,C 180,E1 -6946.198,E2 -6946.198} C_VEL
LIN {X 0,Y 482.243,Z 268.518,A -85,B 0,C 180,E1 -6946.54,E2 -6946.54} C_VEL
LIN {X 0,Y 482.796,Z 251.981,A -85,B 0,C 180,E1 -6949.351,E2 -6949.351} C_VEL
LIN {X 0,Y 483.381,Z 236.647,A -85,B 0,C 180,E1 -6951.986,E2 -6951.986} C_VEL
LIN {X 0,Y 483.458,Z 229.215,A -85,B 0,C 180,E1 -6953.288,E2 -6953.288} C_VEL
LIN {X 0,Y 481.682,Z 219.487,A -85,B 0,C 180,E1 -6955.134,E2 -6955.134} C_VEL
LIN {X 0,Y 481.693,Z 219.485,A -85,B 0,C 180,E1 -6957.832,E2 -6957.832} C_VEL
LIN {X 0,Y 481.646,Z 219.487,A -85,B 0,C 180,E1 -6960.711,E2 -6960.711} C_VEL
LIN {X 0,Y 481.698,Z 219.484,A -85,B 0,C 180,E1 -6963.733,E2 -6963.733} C_VEL
LIN {X 0,Y 481.621,Z 219.49,A -85,B 0,C 180,E1 -6966.747,E2 -6966.747} C_VEL
LIN {X 0,Y 481.677,Z 219.482,A -85,B 0,C 180,E1 -6969.94,E2 -6969.94} C_VEL
LIN {X 0,Y 481.663,Z 219.49,A -85,B 0,C 180,E1 -6973.297,E2 -6973.297} C_VEL
LIN {X 0,Y 481.658,Z 219.488,A -85,B 0,C 180,E1 -6975.641,E2 -6975.641} C_VEL
LIN {X 0,Y 481.656,Z 219.487,A -85,B 0,C 180,E1 -6978.958,E2 -6978.958} C_VEL
LIN {X 0,Y 481.655,Z 219.483,A -85,B 0,C 180,E1 -6981.992,E2 -6981.992} C_VEL
LIN {X 0,Y 481.692,Z 219.484,A -85,B 0,C 180,E1 -6985.318,E2 -6985.318} C_VEL
LIN {X 0,Y 481.644,Z 219.483,A -85,B 0,C 180,E1 -6988.311,E2 -6988.311} C_VEL
LIN {X 0,Y 481.7,Z 219.483,A -85,B 0,C 180,E1 -6991.218,E2 -6991.218} C_VEL
LIN {X 0,Y 481.7,Z 219.478,A -85,B 0,C 180,E1 -6994.043,E2 -6994.043} C_VEL
LIN {X 0,Y 481.673,Z 219.485,A -85,B 0,C 180,E1 -6996.812,E2 -6996.812} C_VEL
LIN {X 0,Y 481.694,Z 219.481,A -85,B 0,C 180,E1 -6999.503,E2 -6999.503} C_VEL
LIN {X 0,Y 481.703,Z 219.475,A -85,B 0,C 180,E1 -7002.158,E2 -7002.158} C_VEL
LIN {X 0,Y 481.742,Z 219.478,A -85,B 0,C 180,E1 -7004.776,E2 -7004.776} C_VEL
LIN {X 0,Y 481.75,Z 219.472,A -85,B 0,C 180,E1 -7008.215,E2 -7008.215} C_VEL
LIN {X 0,Y 481.762,Z 219.47,A -85,B 0,C 180,E1 -7011.612,E2 -7011.612} C_VEL
LIN {X 0,Y 481.807,Z 219.464,A -85,B 0,C 180,E1 -7014.14,E2 -7014.14} C_VEL
LIN {X 0,Y 481.927,Z 219.451,A -85,B 0,C 180,E1 -7017.493,E2 -7017.493} C_VEL
LIN {X 0,Y 481.904,Z 219.458,A -85,B 0,C 180,E1 -7020.836,E2 -7020.836} C_VEL
LIN {X 0,Y 481.927,Z 219.454,A -85,B 0,C 180,E1 -7022.508,E2 -7022.508} C_VEL
LIN {X 0,Y 481.807,Z 219.465,A -85,B 0,C 180,E1 -7025.861,E2 -7025.861} C_VEL
LIN {X 0,Y 481.762,Z 219.472,A -85,B 0,C 180,E1 -7028.388,E2 -7028.388} C_VEL
LIN {X 0,Y 481.75,Z 219.469,A -85,B 0,C 180,E1 -7031.785,E2 -7031.785} C_VEL
LIN {X 0,Y 481.744,Z 219.473,A -85,B 0,C 180,E1 -7035.224,E2 -7035.224} C_VEL
LIN {X 0,Y 481.711,Z 219.483,A -85,B 0,C 180,E1 -7038.722,E2 -7038.722} C_VEL
LIN {X 0,Y 481.645,Z 219.485,A -85,B 0,C 180,E1 -7041.395,E2 -7041.395} C_VEL
LIN {X 0,Y 481.662,Z 219.485,A -85,B 0,C 180,E1 -7044.114,E2 -7044.114} C_VEL
LIN {X 0,Y 481.694,Z 219.481,A -85,B 0,C 180,E1 -7047.127,E2 -7047.127} C_VEL
LIN {X 0,Y 481.673,Z 219.48,A -85,B 0,C 180,E1 -7049.742,E2 -7049.742} C_VEL
LIN {X 0,Y 481.67,Z 219.488,A -85,B 0,C 180,E1 -7052.675,E2 -7052.675} C_VEL
LIN {X 0,Y 481.628,Z 219.49,A -85,B 0,C 180,E1 -7055.711,E2 -7055.711} C_VEL
LIN {X 0,Y 481.656,Z 219.488,A -85,B 0,C 180,E1 -7058.861,E2 -7058.861} C_VEL
LIN {X 0,Y 481.629,Z 219.493,A -85,B 0,C 180,E1 -7062.163,E2 -7062.163} C_VEL
LIN {X 0,Y 481.682,Z 219.62,A -85,B 0,C 180,E1 -7063.909,E2 -7063.909} C_VEL
LIN {X 0,Y 482.746,Z 226.211,A -85,B 0,C 180,E1 -7065.212,E2 -7065.212} C_VEL
LIN {X 0,Y 482.36,Z 242.636,A -85,B 0,C 180,E1 -7068.307,E2 -7068.307} C_VEL
LIN {X 0,Y 482.36,Z 244.128,A -85,B 0,C 180,E1 -7068.543,E2 -7068.543} C_VEL
LIN {X 0,Y 485.021,Z 258.859,A -85,B 0,C 180,E1 -7068.864,E2 -7068.864} C_VEL
LIN {X 0,Y 484.231,Z 351.974,A -85,B 0,C 180,E1 -7070.285,E2 -7070.285} C_VEL
LIN {X 0,Y 483.978,Z 365.515,A -85,B 0,C 180,E1 -7070.675,E2 -7070.675} C_VEL
LIN {X 0,Y 483.726,Z 376.018,A -85,B 0,C 180,E1 -7071.115,E2 -7071.115} C_VEL
LIN {X 0,Y 483.035,Z 381.461,A -85,B 0,C 180,E1 -7071.374,E2 -7071.374} C_VEL
LIN {X 0,Y 479.904,Z 390.13,A -85,B 0,C 180,E1 -7071.813,E2 -7071.813} C_VEL
LIN {X 0,Y 476.657,Z 398.487,A -85,B 0,C 180,E1 -7072.336,E2 -7072.336} C_VEL
LIN {X 0,Y 475.79,Z 403.317,A -85,B 0,C 180,E1 -7072.723,E2 -7072.723} C_VEL
LIN {X 0,Y 475.299,Z 413.605,A -85,B 0,C 180,E1 -7073.739,E2 -7073.739} C_VEL
LIN {X 0,Y 474.921,Z 421.978,A -85,B 0,C 180,E1 -7074.751,E2 -7074.751} C_VEL
LIN {X 0,Y 474.537,Z 430.667,A -85,B 0,C 180,E1 -7076.035,E2 -7076.035} C_VEL
LIN {X 0,Y 474.283,Z 437.226,A -85,B 0,C 180,E1 -7077.24,E2 -7077.24} C_VEL
LIN {X 0,Y 474.028,Z 443.662,A -85,B 0,C 180,E1 -7078.741,E2 -7078.741} C_VEL
LIN {X 0,Y 473.865,Z 448.434,A -85,B 0,C 180,E1 -7080.208,E2 -7080.208} C_VEL
LIN {X 0,Y 473.717,Z 451.796,A -85,B 0,C 180,E1 -7081.657,E2 -7081.657} C_VEL
LIN {X 0,Y 473.641,Z 453.693,A -85,B 0,C 180,E1 -7082.911,E2 -7082.911} C_VEL
LIN {X 0,Y 473.582,Z 454.842,A -85,B 0,C 180,E1 -7084.509,E2 -7084.509} C_VEL
LIN {X 0,Y 473.575,Z 454.861,A -85,B 0,C 180,E1 -7085.447,E2 -7085.447} C_VEL
LIN {X 0,Y 473.59,Z 453.925,A -85,B 0,C 180,E1 -7086.937,E2 -7086.937} C_VEL
LIN {X 0,Y 473.682,Z 452.106,A -85,B 0,C 180,E1 -7088.227,E2 -7088.227} C_VEL
LIN {X 0,Y 473.856,Z 449.115,A -85,B 0,C 180,E1 -7089.602,E2 -7089.602} C_VEL
LIN {X 0,Y 473.991,Z 445.001,A -85,B 0,C 180,E1 -7090.962,E2 -7090.962} C_VEL
LIN {X 0,Y 474.13,Z 439.664,A -85,B 0,C 180,E1 -7092.31,E2 -7092.31} C_VEL
LIN {X 0,Y 474.427,Z 432.864,A -85,B 0,C 180,E1 -7093.653,E2 -7093.653} C_VEL
LIN {X 0,Y 474.808,Z 424.4,A -85,B 0,C 180,E1 -7094.987,E2 -7094.987} C_VEL
LIN {X 0,Y 475.203,Z 415.728,A -85,B 0,C 180,E1 -7096.094,E2 -7096.094} C_VEL
LIN {X 0,Y 475.631,Z 406.169,A -85,B 0,C 180,E1 -7097.086,E2 -7097.086} C_VEL
LIN {X 0,Y 476.082,Z 395.671,A -85,B 0,C 180,E1 -7097.969,E2 -7097.969} C_VEL
LIN {X 0,Y 476.568,Z 384.254,A -85,B 0,C 180,E1 -7098.732,E2 -7098.732} C_VEL
LIN {X 0,Y 476.903,Z 372.668,A -85,B 0,C 180,E1 -7099.331,E2 -7099.331} C_VEL
LIN {X 0,Y 477.214,Z 359.304,A -85,B 0,C 180,E1 -7099.821,E2 -7099.821} C_VEL
LIN {X 0,Y 477.454,Z 346.127,A -85,B 0,C 180,E1 -7100.122,E2 -7100.122} C_VEL
LIN {X 0,Y 478.101,Z 258.397,A -85,B 0,C 180,E1 -7101.459,E2 -7101.459} C_VEL
LIN {X 0,Y 475.363,Z 244.044,A -85,B 0,C 180,E1 -7101.801,E2 -7101.801} C_VEL
LIN {X 0,Y 475.867,Z 229.615,A -85,B 0,C 180,E1 -7104.704,E2 -7104.704} C_VEL
LIN {X 0,Y 475.397,Z 224.562,A -85,B 0,C 180,E1 -7105.761,E2 -7105.761} C_VEL
LIN {X 0,Y 474.668,Z 220.36,A -85,B 0,C 180,E1 -7106.711,E2 -7106.711} C_VEL
LIN {X 0,Y 474.877,Z 220.336,A -85,B 0,C 180,E1 -7107.455,E2 -7107.455} C_VEL
LIN {X 0,Y 474.883,Z 220.332,A -85,B 0,C 180,E1 -7110,E2 -7110} C_VEL
LIN {X 0,Y 474.877,Z 220.328,A -85,B 0,C 180,E1 -7112.545,E2 -7112.545} C_VEL
LIN {X 0,Y 474.743,Z 220.349,A -85,B 0,C 180,E1 -7115.948,E2 -7115.948} C_VEL
LIN {X 0,Y 474.711,Z 220.349,A -85,B 0,C 180,E1 -7118.514,E2 -7118.514} C_VEL
LIN {X 0,Y 474.707,Z 220.353,A -85,B 0,C 180,E1 -7121.962,E2 -7121.962} C_VEL
LIN {X 0,Y 474.682,Z 220.359,A -85,B 0,C 180,E1 -7125.767,E2 -7125.767} C_VEL
LIN {X 0,Y 474.663,Z 220.357,A -85,B 0,C 180,E1 -7129.01,E2 -7129.01} C_VEL
LIN {X 0,Y 474.59,Z 220.37,A -85,B 0,C 180,E1 -7131.729,E2 -7131.729} C_VEL
LIN {X 0,Y 474.629,Z 220.36,A -85,B 0,C 180,E1 -7134.494,E2 -7134.494} C_VEL
LIN {X 0,Y 474.638,Z 220.362,A -85,B 0,C 180,E1 -7137.323,E2 -7137.323} C_VEL
LIN {X 0,Y 474.603,Z 220.364,A -85,B 0,C 180,E1 -7140.23,E2 -7140.23} C_VEL
LIN {X 0,Y 474.644,Z 220.361,A -85,B 0,C 180,E1 -7143.22,E2 -7143.22} C_VEL
LIN {X 0,Y 474.584,Z 220.366,A -85,B 0,C 180,E1 -7146.323,E2 -7146.323} C_VEL
LIN {X 0,Y 474.613,Z 220.368,A -85,B 0,C 180,E1 -7149.645,E2 -7149.645} C_VEL
LIN {X 0,Y 474.6,Z 220.365,A -85,B 0,C 180,E1 -7152.233,E2 -7152.233} C_VEL
LIN {X 0,Y 474.616,Z 220.365,A -85,B 0,C 180,E1 -7155.297,E2 -7155.297} C_VEL
LIN {X 0,Y 474.619,Z 220.362,A -85,B 0,C 180,E1 -7158.214,E2 -7158.214} C_VEL
LIN {X 0,Y 474.61,Z 220.368,A -85,B 0,C 180,E1 -7161.542,E2 -7161.542} C_VEL
LIN {X 0,Y 474.628,Z 220.363,A -85,B 0,C 180,E1 -7164.726,E2 -7164.726} C_VEL
LIN {X 0,Y 474.634,Z 220.363,A -85,B 0,C 180,E1 -7167.787,E2 -7167.787} C_VEL
LIN {X 0,Y 474.622,Z 220.365,A -85,B 0,C 180,E1 -7170.884,E2 -7170.884} C_VEL
LIN {X 0,Y 474.659,Z 220.361,A -85,B 0,C 180,E1 -7173.628,E2 -7173.628} C_VEL
LIN {X 0,Y 474.634,Z 220.363,A -85,B 0,C 180,E1 -7176.641,E2 -7176.641} C_VEL
LIN {X 0,Y 474.652,Z 220.359,A -85,B 0,C 180,E1 -7180.089,E2 -7180.089} C_VEL
LIN {X 0,Y 474.645,Z 220.363,A -85,B 0,C 180,E1 -7182.774,E2 -7182.774} C_VEL
LIN {X 0,Y 474.646,Z 220.362,A -85,B 0,C 180,E1 -7185.421,E2 -7185.421} C_VEL
LIN {X 0,Y 474.701,Z 220.353,A -85,B 0,C 180,E1 -7188.037,E2 -7188.037} C_VEL
LIN {X 0,Y 474.726,Z 220.353,A -85,B 0,C 180,E1 -7191.486,E2 -7191.486} C_VEL
LIN {X 0,Y 474.778,Z 220.343,A -85,B 0,C 180,E1 -7194.052,E2 -7194.052} C_VEL
LIN {X 0,Y 474.892,Z 220.332,A -85,B 0,C 180,E1 -7197.455,E2 -7197.455} C_VEL
LIN {X 0,Y 474.909,Z 220.327,A -85,B 0,C 180,E1 -7200,E2 -7200} C_VEL
LIN {X 0,Y 474.892,Z 220.331,A -85,B 0,C 180,E1 -7202.545,E2 -7202.545} C_VEL
LIN {X 0,Y 474.778,Z 220.343,A -85,B 0,C 180,E1 -7205.948,E2 -7205.948} C_VEL
LIN {X 0,Y 474.725,Z 220.352,A -85,B 0,C 180,E1 -7208.514,E2 -7208.514} C_VEL
LIN {X 0,Y 474.701,Z 220.352,A -85,B 0,C 180,E1 -7211.962,E2 -7211.962} C_VEL
LIN {X 0,Y 474.697,Z 220.354,A -85,B 0,C 180,E1 -7215.456,E2 -7215.456} C_VEL
LIN {X 0,Y 474.663,Z 220.359,A -85,B 0,C 180,E1 -7219.01,E2 -7219.01} C_VEL
LIN {X 0,Y 474.588,Z 220.366,A -85,B 0,C 180,E1 -7221.729,E2 -7221.729} C_VEL
LIN {X 0,Y 474.657,Z 220.361,A -85,B 0,C 180,E1 -7224.493,E2 -7224.493} C_VEL
LIN {X 0,Y 474.678,Z 220.356,A -85,B 0,C 180,E1 -7227.335,E2 -7227.335} C_VEL
LIN {X 0,Y 474.603,Z 220.366,A -85,B 0,C 180,E1 -7230.23,E2 -7230.23} C_VEL
LIN {X 0,Y 474.641,Z 220.361,A -85,B 0,C 180,E1 -7233.22,E2 -7233.22} C_VEL
LIN {X 0,Y 474.59,Z 220.368,A -85,B 0,C 180,E1 -7236.324,E2 -7236.324} C_VEL
LIN {X 0,Y 474.625,Z 220.361,A -85,B 0,C 180,E1 -7239.648,E2 -7239.648} C_VEL
LIN {X 0,Y 474.613,Z 220.365,A -85,B 0,C 180,E1 -7242.935,E2 -7242.935} C_VEL
LIN {X 0,Y 474.608,Z 220.363,A -85,B 0,C 180,E1 -7245.896,E2 -7245.896} C_VEL
LIN {X 0,Y 474.627,Z 220.362,A -85,B 0,C 180,E1 -7249.041,E2 -7249.041} C_VEL
LIN {X 0,Y 474.607,Z 220.362,A -85,B 0,C 180,E1 -7251.705,E2 -7251.705} C_VEL
LIN {X 0,Y 474.622,Z 220.365,A -85,B 0,C 180,E1 -7254.726,E2 -7254.726} C_VEL
LIN {X 0,Y 474.636,Z 220.358,A -85,B 0,C 180,E1 -7257.788,E2 -7257.788} C_VEL
LIN {X 0,Y 474.623,Z 220.366,A -85,B 0,C 180,E1 -7260.885,E2 -7260.885} C_VEL
LIN {X 0,Y 474.627,Z 220.366,A -85,B 0,C 180,E1 -7263.627,E2 -7263.627} C_VEL
LIN {X 0,Y 474.648,Z 220.528,A -85,B 0,C 180,E1 -7264.584,E2 -7264.584} C_VEL
LIN {X 0,Y 476.606,Z 230.679,A -85,B 0,C 180,E1 -7266.538,E2 -7266.538} C_VEL
LIN {X 0,Y 476.461,Z 239.688,A -85,B 0,C 180,E1 -7268.157,E2 -7268.157} C_VEL
LIN {X 0,Y 475.687,Z 258.564,A -85,B 0,C 180,E1 -7271.479,E2 -7271.479} C_VEL
LIN {X 0,Y 475.282,Z 268.686,A -85,B 0,C 180,E1 -7273.241,E2 -7273.241} C_VEL
LIN {X 0,Y 478.002,Z 285.889,A -85,B 0,C 180,E1 -7273.611,E2 -7273.611} C_VEL
LIN {X 0,Y 477.328,Z 376.923,A -85,B 0,C 180,E1 -7275.014,E2 -7275.014} C_VEL
LIN {X 0,Y 476.999,Z 390.154,A -85,B 0,C 180,E1 -7275.386,E2 -7275.386} C_VEL
LIN {X 0,Y 476.598,Z 402.873,A -85,B 0,C 180,E1 -7275.918,E2 -7275.918} C_VEL
LIN {X 0,Y 476.175,Z 414.179,A -85,B 0,C 180,E1 -7276.559,E2 -7276.559} C_VEL
LIN {X 0,Y 475.674,Z 425.162,A -85,B 0,C 180,E1 -7277.355,E2 -7277.355} C_VEL
LIN {X 0,Y 475.279,Z 435.278,A -85,B 0,C 180,E1 -7278.269,E2 -7278.269} C_VEL
LIN {X 0,Y 474.788,Z 444.935,A -85,B 0,C 180,E1 -7279.337,E2 -7279.337} C_VEL
LIN {X 0,Y 474.457,Z 452.854,A -85,B 0,C 180,E1 -7280.408,E2 -7280.408} C_VEL
LIN {X 0,Y 474.162,Z 460.589,A -85,B 0,C 180,E1 -7281.691,E2 -7281.691} C_VEL
LIN {X 0,Y 473.926,Z 467.707,A -85,B 0,C 180,E1 -7283.187,E2 -7283.187} C_VEL
LIN {X 0,Y 473.844,Z 472.446,A -85,B 0,C 180,E1 -7284.468,E2 -7284.468} C_VEL
LIN {X 0,Y 473.733,Z 476.064,A -85,B 0,C 180,E1 -7285.746,E2 -7285.746} C_VEL
LIN {X 0,Y 473.795,Z 477.933,A -85,B 0,C 180,E1 -7286.599,E2 -7286.599} C_VEL
LIN {X 0,Y 473.741,Z 479.331,A -85,B 0,C 180,E1 -7287.449,E2 -7287.449} C_VEL
LIN {X 0,Y 473.688,Z 480.934,A -85,B 0,C 180,E1 -7289.15,E2 -7289.15} C_VEL
LIN {X 0,Y 473.671,Z 481.149,A -85,B 0,C 180,E1 -7290,E2 -7290} C_VEL
LIN {X 0,Y 473.688,Z 480.93,A -85,B 0,C 180,E1 -7290.85,E2 -7290.85} C_VEL
LIN {X 0,Y 473.741,Z 479.318,A -85,B 0,C 180,E1 -7292.551,E2 -7292.551} C_VEL
LIN {X 0,Y 473.795,Z 477.917,A -85,B 0,C 180,E1 -7293.402,E2 -7293.402} C_VEL
LIN {X 0,Y 473.761,Z 474.967,A -85,B 0,C 180,E1 -7294.68,E2 -7294.68} C_VEL
LIN {X 0,Y 473.832,Z 470.978,A -85,B 0,C 180,E1 -7295.96,E2 -7295.96} C_VEL
LIN {X 0,Y 474.015,Z 464.844,A -85,B 0,C 180,E1 -7297.454,E2 -7297.454} C_VEL
LIN {X 0,Y 474.278,Z 458.144,A -85,B 0,C 180,E1 -7298.736,E2 -7298.736} C_VEL
LIN {X 0,Y 474.577,Z 449.831,A -85,B 0,C 180,E1 -7300.021,E2 -7300.021} C_VEL
LIN {X 0,Y 475.015,Z 441.308,A -85,B 0,C 180,E1 -7301.089,E2 -7301.089} C_VEL
LIN {X 0,Y 475.476,Z 431,A -85,B 0,C 180,E1 -7302.139,E2 -7302.139} C_VEL
LIN {X 0,Y 475.923,Z 419.085,A -85,B 0,C 180,E1 -7303.112,E2 -7303.112} C_VEL
LIN {X 0,Y 476.433,Z 407.002,A -85,B 0,C 180,E1 -7303.869,E2 -7303.869} C_VEL
LIN {X 0,Y 476.873,Z 394.591,A -85,B 0,C 180,E1 -7304.455,E2 -7304.455} C_VEL
LIN {X 0,Y 477.254,Z 381.806,A -85,B 0,C 180,E1 -7304.879,E2 -7304.879} C_VEL
LIN {X 0,Y 477.519,Z 366.533,A -85,B 0,C 180,E1 -7305.171,E2 -7305.171} C_VEL
LIN {X 0,Y 477.946,Z 285.225,A -85,B 0,C 180,E1 -7306.415,E2 -7306.415} C_VEL
LIN {X 0,Y 475.269,Z 268.394,A -85,B 0,C 180,E1 -7306.777,E2 -7306.777} C_VEL
LIN {X 0,Y 475.827,Z 251.98,A -85,B 0,C 180,E1 -7309.612,E2 -7309.612} C_VEL
LIN {X 0,Y 476.503,Z 235.172,A -85,B 0,C 180,E1 -7312.549,E2 -7312.549} C_VEL
LIN {X 0,Y 476.465,Z 230.019,A -85,B 0,C 180,E1 -7313.469,E2 -7313.469} C_VEL
LIN {X 0,Y 474.65,Z 220.364,A -85,B 0,C 180,E1 -7315.321,E2 -7315.321} C_VEL
LIN {X 0,Y 474.642,Z 220.361,A -85,B 0,C 180,E1 -7318.283,E2 -7318.283} C_VEL
LIN {X 0,Y 474.599,Z 220.371,A -85,B 0,C 180,E1 -7321.218,E2 -7321.218} C_VEL
LIN {X 0,Y 474.632,Z 220.361,A -85,B 0,C 180,E1 -7324.241,E2 -7324.241} C_VEL
LIN {X 0,Y 474.585,Z 220.371,A -85,B 0,C 180,E1 -7327.384,E2 -7327.384} C_VEL
LIN {X 0,Y 474.618,Z 220.364,A -85,B 0,C 180,E1 -7329.646,E2 -7329.646} C_VEL
LIN {X 0,Y 474.615,Z 220.364,A -85,B 0,C 180,E1 -7332.934,E2 -7332.934} C_VEL
LIN {X 0,Y 474.609,Z 220.364,A -85,B 0,C 180,E1 -7335.895,E2 -7335.895} C_VEL
LIN {X 0,Y 474.627,Z 220.363,A -85,B 0,C 180,E1 -7339.041,E2 -7339.041} C_VEL
LIN {X 0,Y 474.61,Z 220.363,A -85,B 0,C 180,E1 -7341.704,E2 -7341.704} C_VEL
LIN {X 0,Y 474.629,Z 220.361,A -85,B 0,C 180,E1 -7344.726,E2 -7344.726} C_VEL
LIN {X 0,Y 474.635,Z 220.357,A -85,B 0,C 180,E1 -7347.788,E2 -7347.788} C_VEL
LIN {X 0,Y 474.624,Z 220.364,A -85,B 0,C 180,E1 -7350.884,E2 -7350.884} C_VEL
LIN {X 0,Y 474.66,Z 220.356,A -85,B 0,C 180,E1 -7353.628,E2 -7353.628} C_VEL
LIN {X 0,Y 474.635,Z 220.36,A -85,B 0,C 180,E1 -7356.641,E2 -7356.641} C_VEL
LIN {X 0,Y 474.654,Z 220.355,A -85,B 0,C 180,E1 -7360.09,E2 -7360.09} C_VEL
LIN {X 0,Y 474.647,Z 220.359,A -85,B 0,C 180,E1 -7362.774,E2 -7362.774} C_VEL
LIN {X 0,Y 474.648,Z 220.354,A -85,B 0,C 180,E1 -7365.421,E2 -7365.421} C_VEL
LIN {X 0,Y 474.703,Z 220.349,A -85,B 0,C 180,E1 -7368.038,E2 -7368.038} C_VEL
LIN {X 0,Y 474.727,Z 220.347,A -85,B 0,C 180,E1 -7371.486,E2 -7371.486} C_VEL
LIN {X 0,Y 474.77,Z 220.341,A -85,B 0,C 180,E1 -7374.052,E2 -7374.052} C_VEL
LIN {X 0,Y 474.894,Z 220.327,A -85,B 0,C 180,E1 -7377.455,E2 -7377.455} C_VEL
LIN {X 0,Y 474.911,Z 220.32,A -85,B 0,C 180,E1 -7380,E2 -7380} C_VEL
LIN {X 0,Y 474.893,Z 220.331,A -85,B 0,C 180,E1 -7382.545,E2 -7382.545} C_VEL
LIN {X 0,Y 474.769,Z 220.342,A -85,B 0,C 180,E1 -7385.948,E2 -7385.948} C_VEL
LIN {X 0,Y 474.727,Z 220.349,A -85,B 0,C 180,E1 -7388.514,E2 -7388.514} C_VEL
LIN {X 0,Y 474.703,Z 220.347,A -85,B 0,C 180,E1 -7391.963,E2 -7391.963} C_VEL
LIN {X 0,Y 474.7,Z 220.349,A -85,B 0,C 180,E1 -7395.456,E2 -7395.456} C_VEL
LIN {X 0,Y 474.664,Z 220.359,A -85,B 0,C 180,E1 -7399.01,E2 -7399.01} C_VEL
LIN {X 0,Y 474.588,Z 220.364,A -85,B 0,C 180,E1 -7401.729,E2 -7401.729} C_VEL
LIN {X 0,Y 474.64,Z 220.364,A -85,B 0,C 180,E1 -7404.494,E2 -7404.494} C_VEL
LIN {X 0,Y 474.636,Z 220.36,A -85,B 0,C 180,E1 -7407.324,E2 -7407.324} C_VEL
LIN {X 0,Y 474.602,Z 220.365,A -85,B 0,C 180,E1 -7410.231,E2 -7410.231} C_VEL
LIN {X 0,Y 474.624,Z 220.363,A -85,B 0,C 180,E1 -7413.222,E2 -7413.222} C_VEL
LIN {X 0,Y 474.58,Z 220.374,A -85,B 0,C 180,E1 -7416.325,E2 -7416.325} C_VEL
LIN {X 0,Y 474.601,Z 220.365,A -85,B 0,C 180,E1 -7419.644,E2 -7419.644} C_VEL
LIN {X 0,Y 474.588,Z 220.371,A -85,B 0,C 180,E1 -7422.232,E2 -7422.232} C_VEL
LIN {X 0,Y 474.633,Z 220.398,A -85,B 0,C 180,E1 -7423.705,E2 -7423.705} C_VEL
LIN {X 0,Y 475.805,Z 227.597,A -85,B 0,C 180,E1 -7425.154,E2 -7425.154} C_VEL
LIN {X 0,Y 475.392,Z 244.097,A -85,B 0,C 180,E1 -7428.286,E2 -7428.286} C_VEL
LIN {X 0,Y 478.188,Z 258.672,A -85,B 0,C 180,E1 -7428.617,E2 -7428.617} C_VEL
LIN {X 0,Y 477.394,Z 352.012,A -85,B 0,C 180,E1 -7430.062,E2 -7430.062} C_VEL
LIN {X 0,Y 477.131,Z 365.66,A -85,B 0,C 180,E1 -7430.46,E2 -7430.46} C_VEL
LIN {X 0,Y 476.802,Z 378.031,A -85,B 0,C 180,E1 -7430.995,E2 -7430.995} C_VEL
LIN {X 0,Y 476.321,Z 390.136,A -85,B 0,C 180,E1 -7431.706,E2 -7431.706} C_VEL
LIN {X 0,Y 475.841,Z 401.89,A -85,B 0,C 180,E1 -7432.598,E2 -7432.598} C_VEL
LIN {X 0,Y 475.79,Z 403.317,A -85,B 0,C 180,E1 -7432.723,E2 -7432.723} C_VEL
LIN {X 0,Y 474.943,Z 408.042,A -85,B 0,C 180,E1 -7433.14,E2 -7433.14} C_VEL
LIN {X 0,Y 470.324,Z 418.231,A -85,B 0,C 180,E1 -7434.143,E2 -7434.143} C_VEL
LIN {X 0,Y 468.166,Z 423.658,A -85,B 0,C 180,E1 -7434.8,E2 -7434.8} C_VEL
LIN {X 0,Y 467.78,Z 426.185,A -85,B 0,C 180,E1 -7435.161,E2 -7435.161} C_VEL
LIN {X 0,Y 467.398,Z 434.034,A -85,B 0,C 180,E1 -7436.455,E2 -7436.455} C_VEL
